KUKA KRL program: s1001_1.src

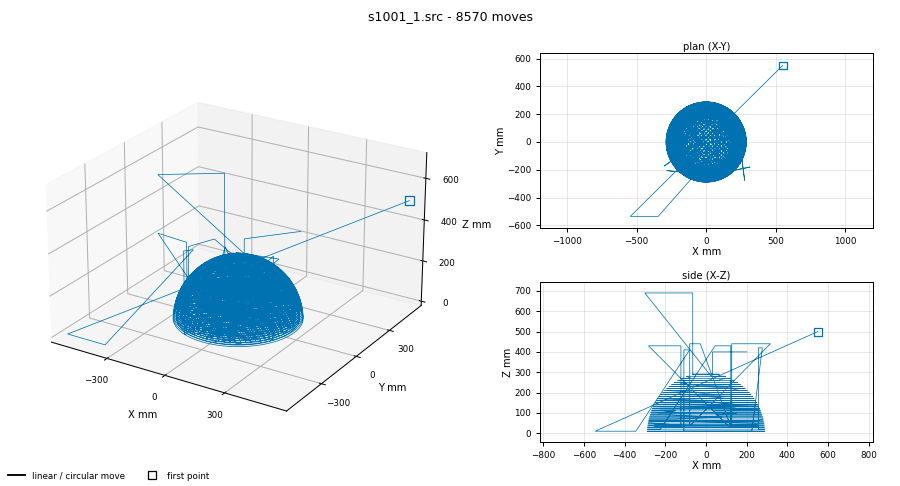
[picture p0: tool path of s1001_1.src, 8570 of 8571 moves have a stored position in this frame; points joined in program order, loops and branches not executed]
&ACCESS RVO
DEF s1001_1()
;TOOLPATH
PTP {A1 0,A2 -135,A3 135,A4 75,A5 30,A6 -65,E1 0,E2 0,E3 0,E4 0,E5 0,E6 0}
$VEL.CP=0.3
LIN {X 550.000,Y 550.000,Z 500.000,A 0.000,B 0.000,C 180.000,E1 0.000} C_DIS
;--------------------------------
;Part 1
;rapid-leaky
LIN {X -545.000,Y -535.000,Z 10.000,A 0.000,B 0.000,C 180.000,E1 0.000} C_DIS

EXTRUDER_STATE=TRUE
LIN {X -545.000,Y -535.000,Z 10.000,A 0.000,B 0.000,C 180.000,E1 0.000} C_DIS
;bead-prime
$VEL.CP=1
LIN {X -345.000,Y -535.000,Z 10.000,A 0.000,B 0.000,C 180.000,E1 0.000} C_DIS
$VEL.CP=0.3
LIN {X -345.000,Y -535.000,Z 10.000,A 0.000,B 0.000,C 180.000,E1 0.000} C_DIS

EXTRUDER_STATE=FALSE
LIN {X -80.274,Y -235.133,Z 410.000,A 0.000,B 0.000,C 180.000,E1 0.000} C_DIS
LIN {X -108.740,Y -267.377,Z 410.000,A 0.000,B 0.000,C 180.000,E1 0.000} C_DIS
LIN {X -108.740,Y -267.377,Z 10.000,A 0.000,B 0.000,C 180.000,E1 0.000} C_DIS
LIN {X -108.740,Y -267.377,Z 10.000,A 0.000,B 0.000,C 180.000,E1 0.000} C_DIS
EXTRUDER_STATE=TRUE

;bead-perimeter_outer
$VEL.CP=0.5
LIN {X -94.832,Y -272.621,Z 10.000,A 0.000,B 0.000,C 180.000,E1 0.000} C_DIS
LIN {X -80.672,Y -277.141,Z 10.000,A 0.000,B 0.000,C 180.000,E1 0.000} C_DIS
LIN {X -66.297,Y -280.927,Z 10.000,A 0.000,B 0.000,C 180.000,E1 0.000} C_DIS
LIN {X -51.748,Y -283.967,Z 10.000,A 0.000,B 0.000,C 180.000,E1 0.000} C_DIS
LIN {X -37.062,Y -286.255,Z 10.000,A 0.000,B 0.000,C 180.000,E1 0.000} C_DIS
LIN {X -22.276,Y -287.783,Z 10.000,A 0.000,B 0.000,C 180.000,E1 0.000} C_DIS
LIN {X -7.431,Y -288.549,Z 10.000,A 0.000,B 0.000,C 180.000,E1 0.000} C_DIS
LIN {X 7.431,Y -288.549,Z 10.000,A 0.000,B 0.000,C 180.000,E1 0.000} C_DIS
LIN {X 22.276,Y -287.783,Z 10.000,A 0.000,B 0.000,C 180.000,E1 0.000} C_DIS
LIN {X 37.062,Y -286.255,Z 10.000,A 0.000,B 0.000,C 180.000,E1 0.000} C_DIS
LIN {X 51.748,Y -283.967,Z 10.000,A 0.000,B 0.000,C 180.000,E1 0.000} C_DIS
LIN {X 66.297,Y -280.927,Z 10.000,A 0.000,B 0.000,C 180.000,E1 0.000} C_DIS
LIN {X 80.672,Y -277.141,Z 10.000,A 0.000,B 0.000,C 180.000,E1 0.000} C_DIS
LIN {X 94.832,Y -272.621,Z 10.000,A 0.000,B 0.000,C 180.000,E1 0.000} C_DIS
LIN {X 108.740,Y -267.377,Z 10.000,A 0.000,B 0.000,C 180.000,E1 0.000} C_DIS
LIN {X 122.360,Y -261.425,Z 10.000,A 0.000,B 0.000,C 180.000,E1 0.000} C_DIS
LIN {X 135.656,Y -254.780,Z 10.000,A 0.000,B 0.000,C 180.000,E1 0.000} C_DIS
LIN {X 148.592,Y -247.459,Z 10.000,A 0.000,B 0.000,C 180.000,E1 0.000} C_DIS
LIN {X 161.134,Y -239.481,Z 10.000,A 0.000,B 0.000,C 180.000,E1 0.000} C_DIS
LIN {X 173.248,Y -230.869,Z 10.000,A 0.000,B 0.000,C 180.000,E1 0.000} C_DIS
LIN {X 184.903,Y -221.644,Z 10.000,A 0.000,B 0.000,C 180.000,E1 0.000} C_DIS
LIN {X 196.068,Y -211.831,Z 10.000,A 0.000,B 0.000,C 180.000,E1 0.000} C_DIS
LIN {X 206.713,Y -201.457,Z 10.000,A 0.000,B 0.000,C 180.000,E1 0.000} C_DIS
LIN {X 216.810,Y -190.549,Z 10.000,A 0.000,B 0.000,C 180.000,E1 0.000} C_DIS
LIN {X 226.331,Y -179.135,Z 10.000,A 0.000,B 0.000,C 180.000,E1 0.000} C_DIS
LIN {X 235.253,Y -167.246,Z 10.000,A 0.000,B 0.000,C 180.000,E1 0.000} C_DIS
LIN {X 243.551,Y -154.914,Z 10.000,A 0.000,B 0.000,C 180.000,E1 0.000} C_DIS
LIN {X 251.203,Y -142.171,Z 10.000,A 0.000,B 0.000,C 180.000,E1 0.000} C_DIS
LIN {X 258.188,Y -129.051,Z 10.000,A 0.000,B 0.000,C 180.000,E1 0.000} C_DIS
LIN {X 264.490,Y -115.588,Z 10.000,A 0.000,B 0.000,C 180.000,E1 0.000} C_DIS
LIN {X 270.089,Y -101.820,Z 10.000,A 0.000,B 0.000,C 180.000,E1 0.000} C_DIS
LIN {X 274.972,Y -87.780,Z 10.000,A 0.000,B 0.000,C 180.000,E1 0.000} C_DIS
LIN {X 279.127,Y -73.509,Z 10.000,A 0.000,B 0.000,C 180.000,E1 0.000} C_DIS
LIN {X 282.541,Y -59.043,Z 10.000,A 0.000,B 0.000,C 180.000,E1 0.000} C_DIS
LIN {X 285.206,Y -44.419,Z 10.000,A 0.000,B 0.000,C 180.000,E1 0.000} C_DIS
LIN {X 287.114,Y -29.678,Z 10.000,A 0.000,B 0.000,C 180.000,E1 0.000} C_DIS
LIN {X 288.261,Y -14.860,Z 10.000,A 0.000,B 0.000,C 180.000,E1 0.000} C_DIS
LIN {X 288.644,Y 0.000,Z 10.000,A 0.000,B 0.000,C 180.000,E1 0.000} C_DIS
LIN {X 288.261,Y 14.859,Z 10.000,A 0.000,B 0.000,C 180.000,E1 0.000} C_DIS
LIN {X 287.114,Y 29.678,Z 10.000,A 0.000,B 0.000,C 180.000,E1 0.000} C_DIS
LIN {X 285.206,Y 44.419,Z 10.000,A 0.000,B 0.000,C 180.000,E1 0.000} C_DIS
LIN {X 282.541,Y 59.043,Z 10.000,A 0.000,B 0.000,C 180.000,E1 0.000} C_DIS
LIN {X 279.127,Y 73.509,Z 10.000,A 0.000,B 0.000,C 180.000,E1 0.000} C_DIS
LIN {X 274.972,Y 87.780,Z 10.000,A 0.000,B 0.000,C 180.000,E1 0.000} C_DIS
LIN {X 270.089,Y 101.820,Z 10.000,A 0.000,B 0.000,C 180.000,E1 0.000} C_DIS
LIN {X 264.490,Y 115.588,Z 10.000,A 0.000,B 0.000,C 180.000,E1 0.000} C_DIS
LIN {X 258.188,Y 129.051,Z 10.000,A 0.000,B 0.000,C 180.000,E1 0.000} C_DIS
LIN {X 251.203,Y 142.171,Z 10.000,A 0.000,B 0.000,C 180.000,E1 0.000} C_DIS
LIN {X 243.551,Y 154.914,Z 10.000,A 0.000,B 0.000,C 180.000,E1 0.000} C_DIS
LIN {X 235.253,Y 167.246,Z 10.000,A 0.000,B 0.000,C 180.000,E1 0.000} C_DIS
LIN {X 226.331,Y 179.135,Z 10.000,A 0.000,B 0.000,C 180.000,E1 0.000} C_DIS
LIN {X 216.810,Y 190.549,Z 10.000,A 0.000,B 0.000,C 180.000,E1 0.000} C_DIS
LIN {X 206.713,Y 201.457,Z 10.000,A 0.000,B 0.000,C 180.000,E1 0.000} C_DIS
LIN {X 196.068,Y 211.831,Z 10.000,A 0.000,B 0.000,C 180.000,E1 0.000} C_DIS
LIN {X 184.903,Y 221.644,Z 10.000,A 0.000,B 0.000,C 180.000,E1 0.000} C_DIS
LIN {X 173.248,Y 230.869,Z 10.000,A 0.000,B 0.000,C 180.000,E1 0.000} C_DIS
LIN {X 161.133,Y 239.482,Z 10.000,A 0.000,B 0.000,C 180.000,E1 0.000} C_DIS
LIN {X 148.592,Y 247.459,Z 10.000,A 0.000,B 0.000,C 180.000,E1 0.000} C_DIS
LIN {X 135.656,Y 254.780,Z 10.000,A 0.000,B 0.000,C 180.000,E1 0.000} C_DIS
LIN {X 122.360,Y 261.425,Z 10.000,A 0.000,B 0.000,C 180.000,E1 0.000} C_DIS
LIN {X 108.740,Y 267.377,Z 10.000,A 0.000,B 0.000,C 180.000,E1 0.000} C_DIS
LIN {X 94.832,Y 272.621,Z 10.000,A 0.000,B 0.000,C 180.000,E1 0.000} C_DIS
LIN {X 80.672,Y 277.141,Z 10.000,A 0.000,B 0.000,C 180.000,E1 0.000} C_DIS
LIN {X 66.297,Y 280.927,Z 10.000,A 0.000,B 0.000,C 180.000,E1 0.000} C_DIS
LIN {X 51.748,Y 283.967,Z 10.000,A 0.000,B 0.000,C 180.000,E1 0.000} C_DIS
LIN {X 37.062,Y 286.255,Z 10.000,A 0.000,B 0.000,C 180.000,E1 0.000} C_DIS
LIN {X 22.276,Y 287.783,Z 10.000,A 0.000,B 0.000,C 180.000,E1 0.000} C_DIS
LIN {X 7.431,Y 288.549,Z 10.000,A 0.000,B 0.000,C 180.000,E1 0.000} C_DIS
LIN {X -7.431,Y 288.549,Z 10.000,A 0.000,B 0.000,C 180.000,E1 0.000} C_DIS
LIN {X -22.276,Y 287.783,Z 10.000,A 0.000,B 0.000,C 180.000,E1 0.000} C_DIS
LIN {X -37.062,Y 286.255,Z 10.000,A 0.000,B 0.000,C 180.000,E1 0.000} C_DIS
LIN {X -51.748,Y 283.967,Z 10.000,A 0.000,B 0.000,C 180.000,E1 0.000} C_DIS
LIN {X -66.297,Y 280.927,Z 10.000,A 0.000,B 0.000,C 180.000,E1 0.000} C_DIS
LIN {X -80.672,Y 277.141,Z 10.000,A 0.000,B 0.000,C 180.000,E1 0.000} C_DIS
LIN {X -94.832,Y 272.621,Z 10.000,A 0.000,B 0.000,C 180.000,E1 0.000} C_DIS
LIN {X -108.740,Y 267.377,Z 10.000,A 0.000,B 0.000,C 180.000,E1 0.000} C_DIS
LIN {X -122.360,Y 261.425,Z 10.000,A 0.000,B 0.000,C 180.000,E1 0.000} C_DIS
LIN {X -135.656,Y 254.780,Z 10.000,A 0.000,B 0.000,C 180.000,E1 0.000} C_DIS
LIN {X -148.592,Y 247.459,Z 10.000,A 0.000,B 0.000,C 180.000,E1 0.000} C_DIS
LIN {X -161.134,Y 239.481,Z 10.000,A 0.000,B 0.000,C 180.000,E1 0.000} C_DIS
LIN {X -173.248,Y 230.869,Z 10.000,A 0.000,B 0.000,C 180.000,E1 0.000} C_DIS
LIN {X -184.903,Y 221.644,Z 10.000,A 0.000,B 0.000,C 180.000,E1 0.000} C_DIS
LIN {X -196.068,Y 211.831,Z 10.000,A 0.000,B 0.000,C 180.000,E1 0.000} C_DIS
LIN {X -206.713,Y 201.457,Z 10.000,A 0.000,B 0.000,C 180.000,E1 0.000} C_DIS
LIN {X -216.810,Y 190.549,Z 10.000,A 0.000,B 0.000,C 180.000,E1 0.000} C_DIS
LIN {X -226.331,Y 179.135,Z 10.000,A 0.000,B 0.000,C 180.000,E1 0.000} C_DIS
LIN {X -235.253,Y 167.246,Z 10.000,A 0.000,B 0.000,C 180.000,E1 0.000} C_DIS
LIN {X -243.551,Y 154.914,Z 10.000,A 0.000,B 0.000,C 180.000,E1 0.000} C_DIS
LIN {X -251.203,Y 142.171,Z 10.000,A 0.000,B 0.000,C 180.000,E1 0.000} C_DIS
LIN {X -258.188,Y 129.051,Z 10.000,A 0.000,B 0.000,C 180.000,E1 0.000} C_DIS
LIN {X -264.490,Y 115.588,Z 10.000,A 0.000,B 0.000,C 180.000,E1 0.000} C_DIS
LIN {X -270.089,Y 101.820,Z 10.000,A 0.000,B 0.000,C 180.000,E1 0.000} C_DIS
LIN {X -274.972,Y 87.780,Z 10.000,A 0.000,B 0.000,C 180.000,E1 0.000} C_DIS
LIN {X -279.127,Y 73.509,Z 10.000,A 0.000,B 0.000,C 180.000,E1 0.000} C_DIS
LIN {X -282.541,Y 59.043,Z 10.000,A 0.000,B 0.000,C 180.000,E1 0.000} C_DIS
LIN {X -285.206,Y 44.419,Z 10.000,A 0.000,B 0.000,C 180.000,E1 0.000} C_DIS
LIN {X -287.114,Y 29.678,Z 10.000,A 0.000,B 0.000,C 180.000,E1 0.000} C_DIS
LIN {X -287.873,Y 19.878,Z 10.000,A 0.000,B 0.000,C 180.000,E1 0.000} C_DIS
LIN {X -288.261,Y 14.860,Z 10.000,A 0.000,B 0.000,C 180.000,E1 0.000} C_DIS
LIN {X -288.644,Y 0.000,Z 10.000,A 0.000,B 0.000,C 180.000,E1 0.000} C_DIS
LIN {X -288.261,Y -14.859,Z 10.000,A 0.000,B 0.000,C 180.000,E1 0.000} C_DIS
LIN {X -287.114,Y -29.678,Z 10.000,A 0.000,B 0.000,C 180.000,E1 0.000} C_DIS
LIN {X -285.206,Y -44.419,Z 10.000,A 0.000,B 0.000,C 180.000,E1 0.000} C_DIS
LIN {X -282.541,Y -59.043,Z 10.000,A 0.000,B 0.000,C 180.000,E1 0.000} C_DIS
LIN {X -279.127,Y -73.509,Z 10.000,A 0.000,B 0.000,C 180.000,E1 0.000} C_DIS
LIN {X -274.972,Y -87.780,Z 10.000,A 0.000,B 0.000,C 180.000,E1 0.000} C_DIS
LIN {X -270.089,Y -101.820,Z 10.000,A 0.000,B 0.000,C 180.000,E1 0.000} C_DIS
LIN {X -264.490,Y -115.588,Z 10.000,A 0.000,B 0.000,C 180.000,E1 0.000} C_DIS
LIN {X -258.188,Y -129.051,Z 10.000,A 0.000,B 0.000,C 180.000,E1 0.000} C_DIS
LIN {X -251.203,Y -142.171,Z 10.000,A 0.000,B 0.000,C 180.000,E1 0.000} C_DIS
LIN {X -243.551,Y -154.914,Z 10.000,A 0.000,B 0.000,C 180.000,E1 0.000} C_DIS
LIN {X -235.253,Y -167.246,Z 10.000,A 0.000,B 0.000,C 180.000,E1 0.000} C_DIS
LIN {X -226.331,Y -179.135,Z 10.000,A 0.000,B 0.000,C 180.000,E1 0.000} C_DIS
LIN {X -216.810,Y -190.549,Z 10.000,A 0.000,B 0.000,C 180.000,E1 0.000} C_DIS
LIN {X -206.713,Y -201.457,Z 10.000,A 0.000,B 0.000,C 180.000,E1 0.000} C_DIS
LIN {X -196.068,Y -211.831,Z 10.000,A 0.000,B 0.000,C 180.000,E1 0.000} C_DIS
LIN {X -184.903,Y -221.644,Z 10.000,A 0.000,B 0.000,C 180.000,E1 0.000} C_DIS
LIN {X -173.248,Y -230.869,Z 10.000,A 0.000,B 0.000,C 180.000,E1 0.000} C_DIS
LIN {X -161.133,Y -239.482,Z 10.000,A 0.000,B 0.000,C 180.000,E1 0.000} C_DIS
LIN {X -148.592,Y -247.459,Z 10.000,A 0.000,B 0.000,C 180.000,E1 0.000} C_DIS
LIN {X -135.656,Y -254.780,Z 10.000,A 0.000,B 0.000,C 180.000,E1 0.000} C_DIS
LIN {X -122.360,Y -261.425,Z 10.000,A 0.000,B 0.000,C 180.000,E1 0.000} C_DIS
LIN {X -108.740,Y -267.377,Z 10.000,A 0.000,B 0.000,C 180.000,E1 0.000} C_DIS
;rapid-leaky
$VEL.CP=0.3
LIN {X -102.884,Y -252.978,Z 10.000,A 0.000,B 0.000,C 180.000,E1 0.000} C_DIS
;bead-perimeter_inner
$VEL.CP=0.5
LIN {X -89.725,Y -257.938,Z 10.000,A 0.000,B 0.000,C 180.000,E1 0.000} C_DIS
LIN {X -76.327,Y -262.215,Z 10.000,A 0.000,B 0.000,C 180.000,E1 0.000} C_DIS
LIN {X -62.727,Y -265.798,Z 10.000,A 0.000,B 0.000,C 180.000,E1 0.000} C_DIS
LIN {X -48.961,Y -268.674,Z 10.000,A 0.000,B 0.000,C 180.000,E1 0.000} C_DIS
LIN {X -35.066,Y -270.839,Z 10.000,A 0.000,B 0.000,C 180.000,E1 0.000} C_DIS
LIN {X -21.076,Y -272.284,Z 10.000,A 0.000,B 0.000,C 180.000,E1 0.000} C_DIS
LIN {X -7.030,Y -273.009,Z 10.000,A 0.000,B 0.000,C 180.000,E1 0.000} C_DIS
LIN {X 7.030,Y -273.009,Z 10.000,A 0.000,B 0.000,C 180.000,E1 0.000} C_DIS
LIN {X 21.076,Y -272.284,Z 10.000,A 0.000,B 0.000,C 180.000,E1 0.000} C_DIS
LIN {X 35.066,Y -270.839,Z 10.000,A 0.000,B 0.000,C 180.000,E1 0.000} C_DIS
LIN {X 48.961,Y -268.674,Z 10.000,A 0.000,B 0.000,C 180.000,E1 0.000} C_DIS
LIN {X 62.727,Y -265.798,Z 10.000,A 0.000,B 0.000,C 180.000,E1 0.000} C_DIS
LIN {X 76.327,Y -262.215,Z 10.000,A 0.000,B 0.000,C 180.000,E1 0.000} C_DIS
LIN {X 89.725,Y -257.938,Z 10.000,A 0.000,B 0.000,C 180.000,E1 0.000} C_DIS
LIN {X 102.884,Y -252.978,Z 10.000,A 0.000,B 0.000,C 180.000,E1 0.000} C_DIS
LIN {X 115.771,Y -247.346,Z 10.000,A 0.000,B 0.000,C 180.000,E1 0.000} C_DIS
LIN {X 128.350,Y -241.059,Z 10.000,A 0.000,B 0.000,C 180.000,E1 0.000} C_DIS
LIN {X 140.590,Y -234.132,Z 10.000,A 0.000,B 0.000,C 180.000,E1 0.000} C_DIS
LIN {X 152.456,Y -226.584,Z 10.000,A 0.000,B 0.000,C 180.000,E1 0.000} C_DIS
LIN {X 163.917,Y -218.436,Z 10.000,A 0.000,B 0.000,C 180.000,E1 0.000} C_DIS
LIN {X 174.944,Y -209.707,Z 10.000,A 0.000,B 0.000,C 180.000,E1 0.000} C_DIS
LIN {X 185.508,Y -200.423,Z 10.000,A 0.000,B 0.000,C 180.000,E1 0.000} C_DIS
LIN {X 195.581,Y -190.607,Z 10.000,A 0.000,B 0.000,C 180.000,E1 0.000} C_DIS
LIN {X 205.133,Y -180.287,Z 10.000,A 0.000,B 0.000,C 180.000,E1 0.000} C_DIS
LIN {X 214.142,Y -169.487,Z 10.000,A 0.000,B 0.000,C 180.000,E1 0.000} C_DIS
LIN {X 222.584,Y -158.239,Z 10.000,A 0.000,B 0.000,C 180.000,E1 0.000} C_DIS
LIN {X 230.434,Y -146.571,Z 10.000,A 0.000,B 0.000,C 180.000,E1 0.000} C_DIS
LIN {X 237.674,Y -134.515,Z 10.000,A 0.000,B 0.000,C 180.000,E1 0.000} C_DIS
LIN {X 244.283,Y -122.100,Z 10.000,A 0.000,B 0.000,C 180.000,E1 0.000} C_DIS
LIN {X 250.245,Y -109.363,Z 10.000,A 0.000,B 0.000,C 180.000,E1 0.000} C_DIS
LIN {X 255.543,Y -96.337,Z 10.000,A 0.000,B 0.000,C 180.000,E1 0.000} C_DIS
LIN {X 260.163,Y -83.053,Z 10.000,A 0.000,B 0.000,C 180.000,E1 0.000} C_DIS
LIN {X 264.094,Y -69.550,Z 10.000,A 0.000,B 0.000,C 180.000,E1 0.000} C_DIS
LIN {X 267.325,Y -55.863,Z 10.000,A 0.000,B 0.000,C 180.000,E1 0.000} C_DIS
LIN {X 269.846,Y -42.027,Z 10.000,A 0.000,B 0.000,C 180.000,E1 0.000} C_DIS
LIN {X 271.651,Y -28.079,Z 10.000,A 0.000,B 0.000,C 180.000,E1 0.000} C_DIS
LIN {X 272.737,Y -14.060,Z 10.000,A 0.000,B 0.000,C 180.000,E1 0.000} C_DIS
LIN {X 273.099,Y 0.000,Z 10.000,A 0.000,B 0.000,C 180.000,E1 0.000} C_DIS
LIN {X 272.737,Y 14.059,Z 10.000,A 0.000,B 0.000,C 180.000,E1 0.000} C_DIS
LIN {X 271.651,Y 28.080,Z 10.000,A 0.000,B 0.000,C 180.000,E1 0.000} C_DIS
LIN {X 269.846,Y 42.027,Z 10.000,A 0.000,B 0.000,C 180.000,E1 0.000} C_DIS
LIN {X 267.325,Y 55.863,Z 10.000,A 0.000,B 0.000,C 180.000,E1 0.000} C_DIS
LIN {X 264.094,Y 69.550,Z 10.000,A 0.000,B 0.000,C 180.000,E1 0.000} C_DIS
LIN {X 260.163,Y 83.053,Z 10.000,A 0.000,B 0.000,C 180.000,E1 0.000} C_DIS
LIN {X 255.543,Y 96.337,Z 10.000,A 0.000,B 0.000,C 180.000,E1 0.000} C_DIS
LIN {X 250.245,Y 109.363,Z 10.000,A 0.000,B 0.000,C 180.000,E1 0.000} C_DIS
LIN {X 244.283,Y 122.100,Z 10.000,A 0.000,B 0.000,C 180.000,E1 0.000} C_DIS
LIN {X 237.674,Y 134.515,Z 10.000,A 0.000,B 0.000,C 180.000,E1 0.000} C_DIS
LIN {X 230.434,Y 146.571,Z 10.000,A 0.000,B 0.000,C 180.000,E1 0.000} C_DIS
LIN {X 222.584,Y 158.239,Z 10.000,A 0.000,B 0.000,C 180.000,E1 0.000} C_DIS
LIN {X 214.142,Y 169.487,Z 10.000,A 0.000,B 0.000,C 180.000,E1 0.000} C_DIS
LIN {X 205.133,Y 180.287,Z 10.000,A 0.000,B 0.000,C 180.000,E1 0.000} C_DIS
LIN {X 195.581,Y 190.607,Z 10.000,A 0.000,B 0.000,C 180.000,E1 0.000} C_DIS
LIN {X 185.508,Y 200.423,Z 10.000,A 0.000,B 0.000,C 180.000,E1 0.000} C_DIS
LIN {X 174.944,Y 209.707,Z 10.000,A 0.000,B 0.000,C 180.000,E1 0.000} C_DIS
LIN {X 163.918,Y 218.436,Z 10.000,A 0.000,B 0.000,C 180.000,E1 0.000} C_DIS
LIN {X 152.456,Y 226.584,Z 10.000,A 0.000,B 0.000,C 180.000,E1 0.000} C_DIS
LIN {X 140.590,Y 234.132,Z 10.000,A 0.000,B 0.000,C 180.000,E1 0.000} C_DIS
LIN {X 128.350,Y 241.059,Z 10.000,A 0.000,B 0.000,C 180.000,E1 0.000} C_DIS
LIN {X 115.771,Y 247.346,Z 10.000,A 0.000,B 0.000,C 180.000,E1 0.000} C_DIS
LIN {X 102.884,Y 252.978,Z 10.000,A 0.000,B 0.000,C 180.000,E1 0.000} C_DIS
LIN {X 89.725,Y 257.938,Z 10.000,A 0.000,B 0.000,C 180.000,E1 0.000} C_DIS
LIN {X 76.327,Y 262.215,Z 10.000,A 0.000,B 0.000,C 180.000,E1 0.000} C_DIS
LIN {X 62.727,Y 265.798,Z 10.000,A 0.000,B 0.000,C 180.000,E1 0.000} C_DIS
LIN {X 48.961,Y 268.674,Z 10.000,A 0.000,B 0.000,C 180.000,E1 0.000} C_DIS
LIN {X 35.066,Y 270.839,Z 10.000,A 0.000,B 0.000,C 180.000,E1 0.000} C_DIS
LIN {X 21.076,Y 272.284,Z 10.000,A 0.000,B 0.000,C 180.000,E1 0.000} C_DIS
LIN {X 7.030,Y 273.009,Z 10.000,A 0.000,B 0.000,C 180.000,E1 0.000} C_DIS
LIN {X -7.030,Y 273.009,Z 10.000,A 0.000,B 0.000,C 180.000,E1 0.000} C_DIS
LIN {X -21.076,Y 272.284,Z 10.000,A 0.000,B 0.000,C 180.000,E1 0.000} C_DIS
LIN {X -35.066,Y 270.839,Z 10.000,A 0.000,B 0.000,C 180.000,E1 0.000} C_DIS
LIN {X -48.961,Y 268.674,Z 10.000,A 0.000,B 0.000,C 180.000,E1 0.000} C_DIS
LIN {X -62.727,Y 265.798,Z 10.000,A 0.000,B 0.000,C 180.000,E1 0.000} C_DIS
LIN {X -76.327,Y 262.215,Z 10.000,A 0.000,B 0.000,C 180.000,E1 0.000} C_DIS
LIN {X -89.725,Y 257.938,Z 10.000,A 0.000,B 0.000,C 180.000,E1 0.000} C_DIS
LIN {X -102.884,Y 252.978,Z 10.000,A 0.000,B 0.000,C 180.000,E1 0.000} C_DIS
LIN {X -115.771,Y 247.346,Z 10.000,A 0.000,B 0.000,C 180.000,E1 0.000} C_DIS
LIN {X -128.350,Y 241.059,Z 10.000,A 0.000,B 0.000,C 180.000,E1 0.000} C_DIS
LIN {X -140.590,Y 234.132,Z 10.000,A 0.000,B 0.000,C 180.000,E1 0.000} C_DIS
LIN {X -152.456,Y 226.584,Z 10.000,A 0.000,B 0.000,C 180.000,E1 0.000} C_DIS
LIN {X -163.917,Y 218.436,Z 10.000,A 0.000,B 0.000,C 180.000,E1 0.000} C_DIS
LIN {X -174.944,Y 209.707,Z 10.000,A 0.000,B 0.000,C 180.000,E1 0.000} C_DIS
LIN {X -185.508,Y 200.423,Z 10.000,A 0.000,B 0.000,C 180.000,E1 0.000} C_DIS
LIN {X -195.581,Y 190.607,Z 10.000,A 0.000,B 0.000,C 180.000,E1 0.000} C_DIS
LIN {X -205.133,Y 180.287,Z 10.000,A 0.000,B 0.000,C 180.000,E1 0.000} C_DIS
LIN {X -214.142,Y 169.487,Z 10.000,A 0.000,B 0.000,C 180.000,E1 0.000} C_DIS
LIN {X -222.584,Y 158.239,Z 10.000,A 0.000,B 0.000,C 180.000,E1 0.000} C_DIS
LIN {X -230.434,Y 146.571,Z 10.000,A 0.000,B 0.000,C 180.000,E1 0.000} C_DIS
LIN {X -237.674,Y 134.515,Z 10.000,A 0.000,B 0.000,C 180.000,E1 0.000} C_DIS
LIN {X -244.283,Y 122.100,Z 10.000,A 0.000,B 0.000,C 180.000,E1 0.000} C_DIS
LIN {X -250.245,Y 109.363,Z 10.000,A 0.000,B 0.000,C 180.000,E1 0.000} C_DIS
LIN {X -255.543,Y 96.337,Z 10.000,A 0.000,B 0.000,C 180.000,E1 0.000} C_DIS
LIN {X -260.163,Y 83.053,Z 10.000,A 0.000,B 0.000,C 180.000,E1 0.000} C_DIS
LIN {X -264.094,Y 69.550,Z 10.000,A 0.000,B 0.000,C 180.000,E1 0.000} C_DIS
LIN {X -267.325,Y 55.863,Z 10.000,A 0.000,B 0.000,C 180.000,E1 0.000} C_DIS
LIN {X -269.846,Y 42.027,Z 10.000,A 0.000,B 0.000,C 180.000,E1 0.000} C_DIS
LIN {X -271.651,Y 28.079,Z 10.000,A 0.000,B 0.000,C 180.000,E1 0.000} C_DIS
LIN {X -272.380,Y 18.678,Z 10.000,A 0.000,B 0.000,C 180.000,E1 0.000} C_DIS
LIN {X -272.737,Y 14.060,Z 10.000,A 0.000,B 0.000,C 180.000,E1 0.000} C_DIS
LIN {X -273.099,Y 0.000,Z 10.000,A 0.000,B 0.000,C 180.000,E1 0.000} C_DIS
LIN {X -272.737,Y -14.059,Z 10.000,A 0.000,B 0.000,C 180.000,E1 0.000} C_DIS
LIN {X -271.651,Y -28.080,Z 10.000,A 0.000,B 0.000,C 180.000,E1 0.000} C_DIS
LIN {X -269.846,Y -42.027,Z 10.000,A 0.000,B 0.000,C 180.000,E1 0.000} C_DIS
LIN {X -267.325,Y -55.863,Z 10.000,A 0.000,B 0.000,C 180.000,E1 0.000} C_DIS
LIN {X -264.094,Y -69.550,Z 10.000,A 0.000,B 0.000,C 180.000,E1 0.000} C_DIS
LIN {X -260.163,Y -83.053,Z 10.000,A 0.000,B 0.000,C 180.000,E1 0.000} C_DIS
LIN {X -255.543,Y -96.337,Z 10.000,A 0.000,B 0.000,C 180.000,E1 0.000} C_DIS
LIN {X -250.245,Y -109.363,Z 10.000,A 0.000,B 0.000,C 180.000,E1 0.000} C_DIS
LIN {X -244.283,Y -122.100,Z 10.000,A 0.000,B 0.000,C 180.000,E1 0.000} C_DIS
LIN {X -237.674,Y -134.515,Z 10.000,A 0.000,B 0.000,C 180.000,E1 0.000} C_DIS
LIN {X -230.434,Y -146.571,Z 10.000,A 0.000,B 0.000,C 180.000,E1 0.000} C_DIS
LIN {X -222.584,Y -158.239,Z 10.000,A 0.000,B 0.000,C 180.000,E1 0.000} C_DIS
LIN {X -214.142,Y -169.487,Z 10.000,A 0.000,B 0.000,C 180.000,E1 0.000} C_DIS
LIN {X -205.133,Y -180.287,Z 10.000,A 0.000,B 0.000,C 180.000,E1 0.000} C_DIS
LIN {X -195.581,Y -190.607,Z 10.000,A 0.000,B 0.000,C 180.000,E1 0.000} C_DIS
LIN {X -185.508,Y -200.423,Z 10.000,A 0.000,B 0.000,C 180.000,E1 0.000} C_DIS
LIN {X -174.944,Y -209.707,Z 10.000,A 0.000,B 0.000,C 180.000,E1 0.000} C_DIS
LIN {X -163.918,Y -218.436,Z 10.000,A 0.000,B 0.000,C 180.000,E1 0.000} C_DIS
LIN {X -152.456,Y -226.584,Z 10.000,A 0.000,B 0.000,C 180.000,E1 0.000} C_DIS
LIN {X -140.590,Y -234.132,Z 10.000,A 0.000,B 0.000,C 180.000,E1 0.000} C_DIS
LIN {X -128.350,Y -241.059,Z 10.000,A 0.000,B 0.000,C 180.000,E1 0.000} C_DIS
LIN {X -115.771,Y -247.346,Z 10.000,A 0.000,B 0.000,C 180.000,E1 0.000} C_DIS
LIN {X -102.884,Y -252.978,Z 10.000,A 0.000,B 0.000,C 180.000,E1 0.000} C_DIS
;rapid-leaky
$VEL.CP=0.3
LIN {X -225.167,Y -120.215,Z 10.000,A 0.000,B 0.000,C 180.000,E1 0.000} C_DIS
;bead-solid_infill
$VEL.CP=0.5
LIN {X -120.009,Y -225.372,Z 10.000,A 0.000,B 0.000,C 180.000,E1 0.000} C_DIS
LIN {X -120.000,Y -225.377,Z 10.000,A 0.000,B 0.000,C 180.000,E1 0.000} C_DIS
LIN {X -108.240,Y -231.255,Z 10.000,A 0.000,B 0.000,C 180.000,E1 0.000} C_DIS
LIN {X -96.191,Y -236.521,Z 10.000,A 0.000,B 0.000,C 180.000,E1 0.000} C_DIS
LIN {X -83.888,Y -241.159,Z 10.000,A 0.000,B 0.000,C 180.000,E1 0.000} C_DIS
LIN {X -71.361,Y -245.157,Z 10.000,A 0.000,B 0.000,C 180.000,E1 0.000} C_DIS
LIN {X -67.922,Y -246.063,Z 10.000,A 0.000,B 0.000,C 180.000,E1 0.000} C_DIS
LIN {X -246.073,Y -67.912,Z 10.000,A 0.000,B 0.000,C 180.000,E1 0.000} C_DIS
LIN {X -246.914,Y -65.025,Z 10.000,A 0.000,B 0.000,C 180.000,E1 0.000} C_DIS
LIN {X -249.934,Y -52.229,Z 10.000,A 0.000,B 0.000,C 180.000,E1 0.000} C_DIS
LIN {X -252.291,Y -39.293,Z 10.000,A 0.000,B 0.000,C 180.000,E1 0.000} C_DIS
LIN {X -253.629,Y -28.961,Z 10.000,A 0.000,B 0.000,C 180.000,E1 0.000} C_DIS
LIN {X -28.977,Y -253.613,Z 10.000,A 0.000,B 0.000,C 180.000,E1 0.000} C_DIS
LIN {X -19.705,Y -254.571,Z 10.000,A 0.000,B 0.000,C 180.000,E1 0.000} C_DIS
LIN {X -6.571,Y -255.249,Z 10.000,A 0.000,B 0.000,C 180.000,E1 0.000} C_DIS
LIN {X 4.054,Y -255.249,Z 10.000,A 0.000,B 0.000,C 180.000,E1 0.000} C_DIS
LIN {X -255.229,Y 4.034,Z 10.000,A 0.000,B 0.000,C 180.000,E1 0.000} C_DIS
LIN {X -254.994,Y 13.146,Z 10.000,A 0.000,B 0.000,C 180.000,E1 0.000} C_DIS
LIN {X -254.673,Y 17.303,Z 10.000,A 0.000,B 0.000,C 180.000,E1 0.000} C_DIS
LIN {X -253.980,Y 26.252,Z 10.000,A 0.000,B 0.000,C 180.000,E1 0.000} C_DIS
LIN {X -253.071,Y 33.272,Z 10.000,A 0.000,B 0.000,C 180.000,E1 0.000} C_DIS
LIN {X 33.335,Y -253.134,Z 10.000,A 0.000,B 0.000,C 180.000,E1 0.000} C_DIS
LIN {X 45.776,Y -251.196,Z 10.000,A 0.000,B 0.000,C 180.000,E1 0.000} C_DIS
LIN {X 58.646,Y -248.507,Z 10.000,A 0.000,B 0.000,C 180.000,E1 0.000} C_DIS
LIN {X 59.800,Y -248.203,Z 10.000,A 0.000,B 0.000,C 180.000,E1 0.000} C_DIS
LIN {X -248.158,Y 59.754,Z 10.000,A 0.000,B 0.000,C 180.000,E1 0.000} C_DIS
LIN {X -246.914,Y 65.025,Z 10.000,A 0.000,B 0.000,C 180.000,E1 0.000} C_DIS
LIN {X -243.239,Y 77.651,Z 10.000,A 0.000,B 0.000,C 180.000,E1 0.000} C_DIS
LIN {X -241.025,Y 84.016,Z 10.000,A 0.000,B 0.000,C 180.000,E1 0.000} C_DIS
LIN {X 84.079,Y -241.087,Z 10.000,A 0.000,B 0.000,C 180.000,E1 0.000} C_DIS
LIN {X 96.191,Y -236.521,Z 10.000,A 0.000,B 0.000,C 180.000,E1 0.000} C_DIS
LIN {X 106.433,Y -232.045,Z 10.000,A 0.000,B 0.000,C 180.000,E1 0.000} C_DIS
LIN {X -232.020,Y 106.407,Z 10.000,A 0.000,B 0.000,C 180.000,E1 0.000} C_DIS
LIN {X -228.392,Y 114.157,Z 10.000,A 0.000,B 0.000,C 180.000,E1 0.000} C_DIS
LIN {X -222.212,Y 125.764,Z 10.000,A 0.000,B 0.000,C 180.000,E1 0.000} C_DIS
LIN {X -221.375,Y 127.158,Z 10.000,A 0.000,B 0.000,C 180.000,E1 0.000} C_DIS
LIN {X 127.127,Y -221.344,Z 10.000,A 0.000,B 0.000,C 180.000,E1 0.000} C_DIS
LIN {X 131.444,Y -218.900,Z 10.000,A 0.000,B 0.000,C 180.000,E1 0.000} C_DIS
LIN {X 142.538,Y -211.844,Z 10.000,A 0.000,B 0.000,C 180.000,E1 0.000} C_DIS
LIN {X 146.328,Y -209.149,Z 10.000,A 0.000,B 0.000,C 180.000,E1 0.000} C_DIS
LIN {X -209.175,Y 146.353,Z 10.000,A 0.000,B 0.000,C 180.000,E1 0.000} C_DIS
LIN {X -208.104,Y 147.945,Z 10.000,A 0.000,B 0.000,C 180.000,E1 0.000} C_DIS
LIN {X -200.212,Y 158.462,Z 10.000,A 0.000,B 0.000,C 180.000,E1 0.000} C_DIS
LIN {X -195.516,Y 164.090,Z 10.000,A 0.000,B 0.000,C 180.000,E1 0.000} C_DIS
LIN {X 164.136,Y -195.562,Z 10.000,A 0.000,B 0.000,C 180.000,E1 0.000} C_DIS
LIN {X 173.441,Y -187.384,Z 10.000,A 0.000,B 0.000,C 180.000,E1 0.000} C_DIS
LIN {X 180.487,Y -180.517,Z 10.000,A 0.000,B 0.000,C 180.000,E1 0.000} C_DIS
LIN {X -180.518,Y 180.487,Z 10.000,A 0.000,B 0.000,C 180.000,E1 0.000} C_DIS
LIN {X -173.441,Y 187.384,Z 10.000,A 0.000,B 0.000,C 180.000,E1 0.000} C_DIS
LIN {X -164.169,Y 195.534,Z 10.000,A 0.000,B 0.000,C 180.000,E1 0.000} C_DIS
LIN {X 195.489,Y -164.123,Z 10.000,A 0.000,B 0.000,C 180.000,E1 0.000} C_DIS
LIN {X 200.212,Y -158.462,Z 10.000,A 0.000,B 0.000,C 180.000,E1 0.000} C_DIS
LIN {X 208.104,Y -147.945,Z 10.000,A 0.000,B 0.000,C 180.000,E1 0.000} C_DIS
LIN {X 209.150,Y -146.390,Z 10.000,A 0.000,B 0.000,C 180.000,E1 0.000} C_DIS
LIN {X -146.364,Y 209.124,Z 10.000,A 0.000,B 0.000,C 180.000,E1 0.000} C_DIS
LIN {X -142.538,Y 211.844,Z 10.000,A 0.000,B 0.000,C 180.000,E1 0.000} C_DIS
LIN {X -131.444,Y 218.900,Z 10.000,A 0.000,B 0.000,C 180.000,E1 0.000} C_DIS
LIN {X -127.166,Y 221.322,Z 10.000,A 0.000,B 0.000,C 180.000,E1 0.000} C_DIS
LIN {X 221.352,Y -127.196,Z 10.000,A 0.000,B 0.000,C 180.000,E1 0.000} C_DIS
LIN {X 222.212,Y -125.764,Z 10.000,A 0.000,B 0.000,C 180.000,E1 0.000} C_DIS
LIN {X 228.392,Y -114.157,Z 10.000,A 0.000,B 0.000,C 180.000,E1 0.000} C_DIS
LIN {X 232.000,Y -106.448,Z 10.000,A 0.000,B 0.000,C 180.000,E1 0.000} C_DIS
LIN {X -106.475,Y 232.026,Z 10.000,A 0.000,B 0.000,C 180.000,E1 0.000} C_DIS
LIN {X -96.191,Y 236.521,Z 10.000,A 0.000,B 0.000,C 180.000,E1 0.000} C_DIS
LIN {X -84.123,Y 241.070,Z 10.000,A 0.000,B 0.000,C 180.000,E1 0.000} C_DIS
LIN {X 241.009,Y -84.061,Z 10.000,A 0.000,B 0.000,C 180.000,E1 0.000} C_DIS
LIN {X 243.239,Y -77.651,Z 10.000,A 0.000,B 0.000,C 180.000,E1 0.000} C_DIS
LIN {X 244.964,Y -71.725,Z 10.000,A 0.000,B 0.000,C 180.000,E1 0.000} C_DIS
LIN {X 246.914,Y -65.025,Z 10.000,A 0.000,B 0.000,C 180.000,E1 0.000} C_DIS
LIN {X 248.146,Y -59.803,Z 10.000,A 0.000,B 0.000,C 180.000,E1 0.000} C_DIS
LIN {X -59.848,Y 248.190,Z 10.000,A 0.000,B 0.000,C 180.000,E1 0.000} C_DIS
LIN {X -58.646,Y 248.507,Z 10.000,A 0.000,B 0.000,C 180.000,E1 0.000} C_DIS
LIN {X -45.776,Y 251.196,Z 10.000,A 0.000,B 0.000,C 180.000,E1 0.000} C_DIS
LIN {X -33.388,Y 253.126,Z 10.000,A 0.000,B 0.000,C 180.000,E1 0.000} C_DIS
LIN {X 253.064,Y -33.325,Z 10.000,A 0.000,B 0.000,C 180.000,E1 0.000} C_DIS
LIN {X 253.980,Y -26.253,Z 10.000,A 0.000,B 0.000,C 180.000,E1 0.000} C_DIS
LIN {X 255.503,Y -6.574,Z 10.000,A 0.000,B 0.000,C 180.000,E1 0.000} C_DIS
LIN {X 255.444,Y -4.310,Z 10.000,A 0.000,B 0.000,C 180.000,E1 0.000} C_DIS
LIN {X -4.115,Y 255.249,Z 10.000,A 0.000,B 0.000,C 180.000,E1 0.000} C_DIS
LIN {X 6.571,Y 255.249,Z 10.000,A 0.000,B 0.000,C 180.000,E1 0.000} C_DIS
LIN {X 19.705,Y 254.571,Z 10.000,A 0.000,B 0.000,C 180.000,E1 0.000} C_DIS
LIN {X 28.909,Y 253.620,Z 10.000,A 0.000,B 0.000,C 180.000,E1 0.000} C_DIS
LIN {X 253.638,Y 28.892,Z 10.000,A 0.000,B 0.000,C 180.000,E1 0.000} C_DIS
LIN {X 252.291,Y 39.293,Z 10.000,A 0.000,B 0.000,C 180.000,E1 0.000} C_DIS
LIN {X 249.934,Y 52.229,Z 10.000,A 0.000,B 0.000,C 180.000,E1 0.000} C_DIS
LIN {X 246.914,Y 65.025,Z 10.000,A 0.000,B 0.000,C 180.000,E1 0.000} C_DIS
LIN {X 246.098,Y 67.827,Z 10.000,A 0.000,B 0.000,C 180.000,E1 0.000} C_DIS
LIN {X 67.840,Y 246.085,Z 10.000,A 0.000,B 0.000,C 180.000,E1 0.000} C_DIS
LIN {X 71.361,Y 245.157,Z 10.000,A 0.000,B 0.000,C 180.000,E1 0.000} C_DIS
LIN {X 83.888,Y 241.159,Z 10.000,A 0.000,B 0.000,C 180.000,E1 0.000} C_DIS
LIN {X 96.191,Y 236.521,Z 10.000,A 0.000,B 0.000,C 180.000,E1 0.000} C_DIS
LIN {X 108.240,Y 231.255,Z 10.000,A 0.000,B 0.000,C 180.000,E1 0.000} C_DIS
LIN {X 119.887,Y 225.434,Z 10.000,A 0.000,B 0.000,C 180.000,E1 0.000} C_DIS
LIN {X 225.236,Y 120.085,Z 10.000,A 0.000,B 0.000,C 180.000,E1 0.000} C_DIS
$VEL.CP=0.3
LIN {X 225.236,Y 120.085,Z 10.000,A 0.000,B 0.000,C 180.000,E1 0.000} C_DIS
EXTRUDER_STATE=FALSE

LIN {X 277.036,Y -276.547,Z 420.000,A 0.000,B 0.000,C 180.000,E1 0.000} C_DIS
LIN {X 257.744,Y -128.829,Z 420.000,A 0.000,B 0.000,C 180.000,E1 0.000} C_DIS
LIN {X 257.744,Y -128.829,Z 20.000,A 0.000,B 0.000,C 180.000,E1 0.000} C_DIS
LIN {X 257.744,Y -128.829,Z 20.000,A 0.000,B 0.000,C 180.000,E1 0.000} C_DIS
EXTRUDER_STATE=TRUE

;bead-perimeter_outer
$VEL.CP=1
LIN {X 264.034,Y -115.390,Z 20.000,A 0.000,B 0.000,C 180.000,E1 0.000} C_DIS
LIN {X 269.624,Y -101.644,Z 20.000,A 0.000,B 0.000,C 180.000,E1 0.000} C_DIS
LIN {X 274.499,Y -87.629,Z 20.000,A 0.000,B 0.000,C 180.000,E1 0.000} C_DIS
LIN {X 278.646,Y -73.382,Z 20.000,A 0.000,B 0.000,C 180.000,E1 0.000} C_DIS
LIN {X 282.054,Y -58.941,Z 20.000,A 0.000,B 0.000,C 180.000,E1 0.000} C_DIS
LIN {X 284.715,Y -44.343,Z 20.000,A 0.000,B 0.000,C 180.000,E1 0.000} C_DIS
LIN {X 286.619,Y -29.627,Z 20.000,A 0.000,B 0.000,C 180.000,E1 0.000} C_DIS
LIN {X 287.765,Y -14.833,Z 20.000,A 0.000,B 0.000,C 180.000,E1 0.000} C_DIS
LIN {X 288.147,Y 0.000,Z 20.000,A 0.000,B 0.000,C 180.000,E1 0.000} C_DIS
LIN {X 287.765,Y 14.833,Z 20.000,A 0.000,B 0.000,C 180.000,E1 0.000} C_DIS
LIN {X 286.619,Y 29.627,Z 20.000,A 0.000,B 0.000,C 180.000,E1 0.000} C_DIS
LIN {X 284.715,Y 44.343,Z 20.000,A 0.000,B 0.000,C 180.000,E1 0.000} C_DIS
LIN {X 282.054,Y 58.941,Z 20.000,A 0.000,B 0.000,C 180.000,E1 0.000} C_DIS
LIN {X 278.646,Y 73.382,Z 20.000,A 0.000,B 0.000,C 180.000,E1 0.000} C_DIS
LIN {X 274.499,Y 87.629,Z 20.000,A 0.000,B 0.000,C 180.000,E1 0.000} C_DIS
LIN {X 269.624,Y 101.644,Z 20.000,A 0.000,B 0.000,C 180.000,E1 0.000} C_DIS
LIN {X 264.034,Y 115.390,Z 20.000,A 0.000,B 0.000,C 180.000,E1 0.000} C_DIS
LIN {X 257.744,Y 128.829,Z 20.000,A 0.000,B 0.000,C 180.000,E1 0.000} C_DIS
LIN {X 250.770,Y 141.926,Z 20.000,A 0.000,B 0.000,C 180.000,E1 0.000} C_DIS
LIN {X 243.131,Y 154.648,Z 20.000,A 0.000,B 0.000,C 180.000,E1 0.000} C_DIS
LIN {X 234.848,Y 166.958,Z 20.000,A 0.000,B 0.000,C 180.000,E1 0.000} C_DIS
LIN {X 232.107,Y 170.611,Z 20.000,A 0.000,B 0.000,C 180.000,E1 0.000} C_DIS
LIN {X 225.942,Y 178.827,Z 20.000,A 0.000,B 0.000,C 180.000,E1 0.000} C_DIS
LIN {X 216.436,Y 190.221,Z 20.000,A 0.000,B 0.000,C 180.000,E1 0.000} C_DIS
LIN {X 206.357,Y 201.110,Z 20.000,A 0.000,B 0.000,C 180.000,E1 0.000} C_DIS
LIN {X 195.730,Y 211.467,Z 20.000,A 0.000,B 0.000,C 180.000,E1 0.000} C_DIS
LIN {X 184.585,Y 221.262,Z 20.000,A 0.000,B 0.000,C 180.000,E1 0.000} C_DIS
LIN {X 172.949,Y 230.472,Z 20.000,A 0.000,B 0.000,C 180.000,E1 0.000} C_DIS
LIN {X 160.857,Y 239.069,Z 20.000,A 0.000,B 0.000,C 180.000,E1 0.000} C_DIS
LIN {X 148.336,Y 247.033,Z 20.000,A 0.000,B 0.000,C 180.000,E1 0.000} C_DIS
LIN {X 135.422,Y 254.341,Z 20.000,A 0.000,B 0.000,C 180.000,E1 0.000} C_DIS
LIN {X 122.150,Y 260.975,Z 20.000,A 0.000,B 0.000,C 180.000,E1 0.000} C_DIS
LIN {X 108.553,Y 266.916,Z 20.000,A 0.000,B 0.000,C 180.000,E1 0.000} C_DIS
LIN {X 94.668,Y 272.152,Z 20.000,A 0.000,B 0.000,C 180.000,E1 0.000} C_DIS
LIN {X 80.533,Y 276.664,Z 20.000,A 0.000,B 0.000,C 180.000,E1 0.000} C_DIS
LIN {X 66.183,Y 280.443,Z 20.000,A 0.000,B 0.000,C 180.000,E1 0.000} C_DIS
LIN {X 51.659,Y 283.478,Z 20.000,A 0.000,B 0.000,C 180.000,E1 0.000} C_DIS
LIN {X 36.997,Y 285.761,Z 20.000,A 0.000,B 0.000,C 180.000,E1 0.000} C_DIS
LIN {X 22.238,Y 287.287,Z 20.000,A 0.000,B 0.000,C 180.000,E1 0.000} C_DIS
LIN {X 7.419,Y 288.052,Z 20.000,A 0.000,B 0.000,C 180.000,E1 0.000} C_DIS
LIN {X -7.419,Y 288.052,Z 20.000,A 0.000,B 0.000,C 180.000,E1 0.000} C_DIS
LIN {X -22.238,Y 287.287,Z 20.000,A 0.000,B 0.000,C 180.000,E1 0.000} C_DIS
LIN {X -36.997,Y 285.761,Z 20.000,A 0.000,B 0.000,C 180.000,E1 0.000} C_DIS
LIN {X -51.660,Y 283.478,Z 20.000,A 0.000,B 0.000,C 180.000,E1 0.000} C_DIS
LIN {X -66.183,Y 280.443,Z 20.000,A 0.000,B 0.000,C 180.000,E1 0.000} C_DIS
LIN {X -80.533,Y 276.664,Z 20.000,A 0.000,B 0.000,C 180.000,E1 0.000} C_DIS
LIN {X -94.668,Y 272.152,Z 20.000,A 0.000,B 0.000,C 180.000,E1 0.000} C_DIS
LIN {X -108.553,Y 266.916,Z 20.000,A 0.000,B 0.000,C 180.000,E1 0.000} C_DIS
LIN {X -122.150,Y 260.975,Z 20.000,A 0.000,B 0.000,C 180.000,E1 0.000} C_DIS
LIN {X -135.422,Y 254.341,Z 20.000,A 0.000,B 0.000,C 180.000,E1 0.000} C_DIS
LIN {X -148.336,Y 247.033,Z 20.000,A 0.000,B 0.000,C 180.000,E1 0.000} C_DIS
LIN {X -160.857,Y 239.069,Z 20.000,A 0.000,B 0.000,C 180.000,E1 0.000} C_DIS
LIN {X -172.949,Y 230.472,Z 20.000,A 0.000,B 0.000,C 180.000,E1 0.000} C_DIS
LIN {X -184.585,Y 221.262,Z 20.000,A 0.000,B 0.000,C 180.000,E1 0.000} C_DIS
LIN {X -195.730,Y 211.467,Z 20.000,A 0.000,B 0.000,C 180.000,E1 0.000} C_DIS
LIN {X -206.357,Y 201.110,Z 20.000,A 0.000,B 0.000,C 180.000,E1 0.000} C_DIS
LIN {X -216.436,Y 190.221,Z 20.000,A 0.000,B 0.000,C 180.000,E1 0.000} C_DIS
LIN {X -225.942,Y 178.827,Z 20.000,A 0.000,B 0.000,C 180.000,E1 0.000} C_DIS
LIN {X -234.848,Y 166.958,Z 20.000,A 0.000,B 0.000,C 180.000,E1 0.000} C_DIS
LIN {X -243.131,Y 154.648,Z 20.000,A 0.000,B 0.000,C 180.000,E1 0.000} C_DIS
LIN {X -250.770,Y 141.926,Z 20.000,A 0.000,B 0.000,C 180.000,E1 0.000} C_DIS
LIN {X -257.744,Y 128.829,Z 20.000,A 0.000,B 0.000,C 180.000,E1 0.000} C_DIS
LIN {X -264.034,Y 115.390,Z 20.000,A 0.000,B 0.000,C 180.000,E1 0.000} C_DIS
LIN {X -269.624,Y 101.644,Z 20.000,A 0.000,B 0.000,C 180.000,E1 0.000} C_DIS
LIN {X -274.499,Y 87.629,Z 20.000,A 0.000,B 0.000,C 180.000,E1 0.000} C_DIS
LIN {X -278.646,Y 73.382,Z 20.000,A 0.000,B 0.000,C 180.000,E1 0.000} C_DIS
LIN {X -282.054,Y 58.941,Z 20.000,A 0.000,B 0.000,C 180.000,E1 0.000} C_DIS
LIN {X -284.715,Y 44.343,Z 20.000,A 0.000,B 0.000,C 180.000,E1 0.000} C_DIS
LIN {X -286.619,Y 29.627,Z 20.000,A 0.000,B 0.000,C 180.000,E1 0.000} C_DIS
LIN {X -287.765,Y 14.833,Z 20.000,A 0.000,B 0.000,C 180.000,E1 0.000} C_DIS
LIN {X -288.147,Y 0.000,Z 20.000,A 0.000,B 0.000,C 180.000,E1 0.000} C_DIS
LIN {X -287.765,Y -14.833,Z 20.000,A 0.000,B 0.000,C 180.000,E1 0.000} C_DIS
LIN {X -286.619,Y -29.627,Z 20.000,A 0.000,B 0.000,C 180.000,E1 0.000} C_DIS
LIN {X -284.715,Y -44.343,Z 20.000,A 0.000,B 0.000,C 180.000,E1 0.000} C_DIS
LIN {X -282.054,Y -58.941,Z 20.000,A 0.000,B 0.000,C 180.000,E1 0.000} C_DIS
LIN {X -278.646,Y -73.382,Z 20.000,A 0.000,B 0.000,C 180.000,E1 0.000} C_DIS
LIN {X -274.499,Y -87.629,Z 20.000,A 0.000,B 0.000,C 180.000,E1 0.000} C_DIS
LIN {X -269.624,Y -101.644,Z 20.000,A 0.000,B 0.000,C 180.000,E1 0.000} C_DIS
LIN {X -264.034,Y -115.390,Z 20.000,A 0.000,B 0.000,C 180.000,E1 0.000} C_DIS
LIN {X -257.744,Y -128.829,Z 20.000,A 0.000,B 0.000,C 180.000,E1 0.000} C_DIS
LIN {X -250.770,Y -141.926,Z 20.000,A 0.000,B 0.000,C 180.000,E1 0.000} C_DIS
LIN {X -243.131,Y -154.648,Z 20.000,A 0.000,B 0.000,C 180.000,E1 0.000} C_DIS
LIN {X -234.848,Y -166.958,Z 20.000,A 0.000,B 0.000,C 180.000,E1 0.000} C_DIS
LIN {X -225.942,Y -178.827,Z 20.000,A 0.000,B 0.000,C 180.000,E1 0.000} C_DIS
LIN {X -216.436,Y -190.221,Z 20.000,A 0.000,B 0.000,C 180.000,E1 0.000} C_DIS
LIN {X -206.357,Y -201.110,Z 20.000,A 0.000,B 0.000,C 180.000,E1 0.000} C_DIS
LIN {X -195.730,Y -211.467,Z 20.000,A 0.000,B 0.000,C 180.000,E1 0.000} C_DIS
LIN {X -184.585,Y -221.262,Z 20.000,A 0.000,B 0.000,C 180.000,E1 0.000} C_DIS
LIN {X -172.949,Y -230.472,Z 20.000,A 0.000,B 0.000,C 180.000,E1 0.000} C_DIS
LIN {X -160.857,Y -239.069,Z 20.000,A 0.000,B 0.000,C 180.000,E1 0.000} C_DIS
LIN {X -148.336,Y -247.033,Z 20.000,A 0.000,B 0.000,C 180.000,E1 0.000} C_DIS
LIN {X -135.422,Y -254.341,Z 20.000,A 0.000,B 0.000,C 180.000,E1 0.000} C_DIS
LIN {X -122.150,Y -260.975,Z 20.000,A 0.000,B 0.000,C 180.000,E1 0.000} C_DIS
LIN {X -108.553,Y -266.916,Z 20.000,A 0.000,B 0.000,C 180.000,E1 0.000} C_DIS
LIN {X -94.668,Y -272.152,Z 20.000,A 0.000,B 0.000,C 180.000,E1 0.000} C_DIS
LIN {X -80.533,Y -276.664,Z 20.000,A 0.000,B 0.000,C 180.000,E1 0.000} C_DIS
LIN {X -66.183,Y -280.443,Z 20.000,A 0.000,B 0.000,C 180.000,E1 0.000} C_DIS
LIN {X -51.659,Y -283.478,Z 20.000,A 0.000,B 0.000,C 180.000,E1 0.000} C_DIS
LIN {X -36.997,Y -285.761,Z 20.000,A 0.000,B 0.000,C 180.000,E1 0.000} C_DIS
LIN {X -22.238,Y -287.287,Z 20.000,A 0.000,B 0.000,C 180.000,E1 0.000} C_DIS
LIN {X -7.419,Y -288.052,Z 20.000,A 0.000,B 0.000,C 180.000,E1 0.000} C_DIS
LIN {X 7.419,Y -288.052,Z 20.000,A 0.000,B 0.000,C 180.000,E1 0.000} C_DIS
LIN {X 22.238,Y -287.287,Z 20.000,A 0.000,B 0.000,C 180.000,E1 0.000} C_DIS
LIN {X 36.997,Y -285.761,Z 20.000,A 0.000,B 0.000,C 180.000,E1 0.000} C_DIS
LIN {X 51.660,Y -283.478,Z 20.000,A 0.000,B 0.000,C 180.000,E1 0.000} C_DIS
LIN {X 66.183,Y -280.443,Z 20.000,A 0.000,B 0.000,C 180.000,E1 0.000} C_DIS
LIN {X 80.533,Y -276.664,Z 20.000,A 0.000,B 0.000,C 180.000,E1 0.000} C_DIS
LIN {X 94.668,Y -272.152,Z 20.000,A 0.000,B 0.000,C 180.000,E1 0.000} C_DIS
LIN {X 108.553,Y -266.916,Z 20.000,A 0.000,B 0.000,C 180.000,E1 0.000} C_DIS
LIN {X 122.150,Y -260.975,Z 20.000,A 0.000,B 0.000,C 180.000,E1 0.000} C_DIS
LIN {X 135.422,Y -254.341,Z 20.000,A 0.000,B 0.000,C 180.000,E1 0.000} C_DIS
LIN {X 148.336,Y -247.033,Z 20.000,A 0.000,B 0.000,C 180.000,E1 0.000} C_DIS
LIN {X 160.857,Y -239.069,Z 20.000,A 0.000,B 0.000,C 180.000,E1 0.000} C_DIS
LIN {X 172.949,Y -230.472,Z 20.000,A 0.000,B 0.000,C 180.000,E1 0.000} C_DIS
LIN {X 184.585,Y -221.262,Z 20.000,A 0.000,B 0.000,C 180.000,E1 0.000} C_DIS
LIN {X 195.730,Y -211.467,Z 20.000,A 0.000,B 0.000,C 180.000,E1 0.000} C_DIS
LIN {X 206.357,Y -201.110,Z 20.000,A 0.000,B 0.000,C 180.000,E1 0.000} C_DIS
LIN {X 216.436,Y -190.221,Z 20.000,A 0.000,B 0.000,C 180.000,E1 0.000} C_DIS
LIN {X 225.942,Y -178.827,Z 20.000,A 0.000,B 0.000,C 180.000,E1 0.000} C_DIS
LIN {X 234.848,Y -166.958,Z 20.000,A 0.000,B 0.000,C 180.000,E1 0.000} C_DIS
LIN {X 243.131,Y -154.648,Z 20.000,A 0.000,B 0.000,C 180.000,E1 0.000} C_DIS
LIN {X 250.770,Y -141.926,Z 20.000,A 0.000,B 0.000,C 180.000,E1 0.000} C_DIS
LIN {X 257.744,Y -128.829,Z 20.000,A 0.000,B 0.000,C 180.000,E1 0.000} C_DIS
;rapid-leaky
$VEL.CP=0.3
LIN {X 243.839,Y -121.878,Z 20.000,A 0.000,B 0.000,C 180.000,E1 0.000} C_DIS
;bead-perimeter_inner
$VEL.CP=1
LIN {X 249.789,Y -109.164,Z 20.000,A 0.000,B 0.000,C 180.000,E1 0.000} C_DIS
LIN {X 255.078,Y -96.160,Z 20.000,A 0.000,B 0.000,C 180.000,E1 0.000} C_DIS
LIN {X 259.690,Y -82.902,Z 20.000,A 0.000,B 0.000,C 180.000,E1 0.000} C_DIS
LIN {X 263.614,Y -69.424,Z 20.000,A 0.000,B 0.000,C 180.000,E1 0.000} C_DIS
LIN {X 266.838,Y -55.761,Z 20.000,A 0.000,B 0.000,C 180.000,E1 0.000} C_DIS
LIN {X 269.355,Y -41.951,Z 20.000,A 0.000,B 0.000,C 180.000,E1 0.000} C_DIS
LIN {X 271.156,Y -28.029,Z 20.000,A 0.000,B 0.000,C 180.000,E1 0.000} C_DIS
LIN {X 272.241,Y -14.032,Z 20.000,A 0.000,B 0.000,C 180.000,E1 0.000} C_DIS
LIN {X 272.602,Y 0.000,Z 20.000,A 0.000,B 0.000,C 180.000,E1 0.000} C_DIS
LIN {X 272.241,Y 14.032,Z 20.000,A 0.000,B 0.000,C 180.000,E1 0.000} C_DIS
LIN {X 271.156,Y 28.029,Z 20.000,A 0.000,B 0.000,C 180.000,E1 0.000} C_DIS
LIN {X 269.355,Y 41.951,Z 20.000,A 0.000,B 0.000,C 180.000,E1 0.000} C_DIS
LIN {X 266.838,Y 55.761,Z 20.000,A 0.000,B 0.000,C 180.000,E1 0.000} C_DIS
LIN {X 263.614,Y 69.424,Z 20.000,A 0.000,B 0.000,C 180.000,E1 0.000} C_DIS
LIN {X 259.690,Y 82.902,Z 20.000,A 0.000,B 0.000,C 180.000,E1 0.000} C_DIS
LIN {X 255.078,Y 96.160,Z 20.000,A 0.000,B 0.000,C 180.000,E1 0.000} C_DIS
LIN {X 249.789,Y 109.164,Z 20.000,A 0.000,B 0.000,C 180.000,E1 0.000} C_DIS
LIN {X 243.839,Y 121.878,Z 20.000,A 0.000,B 0.000,C 180.000,E1 0.000} C_DIS
LIN {X 237.241,Y 134.269,Z 20.000,A 0.000,B 0.000,C 180.000,E1 0.000} C_DIS
LIN {X 230.014,Y 146.305,Z 20.000,A 0.000,B 0.000,C 180.000,E1 0.000} C_DIS
LIN {X 222.178,Y 157.952,Z 20.000,A 0.000,B 0.000,C 180.000,E1 0.000} C_DIS
LIN {X 219.678,Y 161.284,Z 20.000,A 0.000,B 0.000,C 180.000,E1 0.000} C_DIS
LIN {X 213.753,Y 169.179,Z 20.000,A 0.000,B 0.000,C 180.000,E1 0.000} C_DIS
LIN {X 204.759,Y 179.959,Z 20.000,A 0.000,B 0.000,C 180.000,E1 0.000} C_DIS
LIN {X 195.224,Y 190.261,Z 20.000,A 0.000,B 0.000,C 180.000,E1 0.000} C_DIS
LIN {X 185.170,Y 200.059,Z 20.000,A 0.000,B 0.000,C 180.000,E1 0.000} C_DIS
LIN {X 174.627,Y 209.325,Z 20.000,A 0.000,B 0.000,C 180.000,E1 0.000} C_DIS
LIN {X 163.619,Y 218.038,Z 20.000,A 0.000,B 0.000,C 180.000,E1 0.000} C_DIS
LIN {X 152.179,Y 226.171,Z 20.000,A 0.000,B 0.000,C 180.000,E1 0.000} C_DIS
LIN {X 140.333,Y 233.706,Z 20.000,A 0.000,B 0.000,C 180.000,E1 0.000} C_DIS
LIN {X 128.117,Y 240.620,Z 20.000,A 0.000,B 0.000,C 180.000,E1 0.000} C_DIS
LIN {X 115.561,Y 246.896,Z 20.000,A 0.000,B 0.000,C 180.000,E1 0.000} C_DIS
LIN {X 102.697,Y 252.517,Z 20.000,A 0.000,B 0.000,C 180.000,E1 0.000} C_DIS
LIN {X 89.560,Y 257.470,Z 20.000,A 0.000,B 0.000,C 180.000,E1 0.000} C_DIS
LIN {X 76.188,Y 261.738,Z 20.000,A 0.000,B 0.000,C 180.000,E1 0.000} C_DIS
LIN {X 62.613,Y 265.314,Z 20.000,A 0.000,B 0.000,C 180.000,E1 0.000} C_DIS
LIN {X 48.872,Y 268.185,Z 20.000,A 0.000,B 0.000,C 180.000,E1 0.000} C_DIS
LIN {X 35.002,Y 270.345,Z 20.000,A 0.000,B 0.000,C 180.000,E1 0.000} C_DIS
LIN {X 21.037,Y 271.789,Z 20.000,A 0.000,B 0.000,C 180.000,E1 0.000} C_DIS
LIN {X 7.018,Y 272.512,Z 20.000,A 0.000,B 0.000,C 180.000,E1 0.000} C_DIS
LIN {X -7.018,Y 272.512,Z 20.000,A 0.000,B 0.000,C 180.000,E1 0.000} C_DIS
LIN {X -21.037,Y 271.789,Z 20.000,A 0.000,B 0.000,C 180.000,E1 0.000} C_DIS
LIN {X -35.001,Y 270.345,Z 20.000,A 0.000,B 0.000,C 180.000,E1 0.000} C_DIS
LIN {X -48.873,Y 268.185,Z 20.000,A 0.000,B 0.000,C 180.000,E1 0.000} C_DIS
LIN {X -62.613,Y 265.314,Z 20.000,A 0.000,B 0.000,C 180.000,E1 0.000} C_DIS
LIN {X -76.188,Y 261.738,Z 20.000,A 0.000,B 0.000,C 180.000,E1 0.000} C_DIS
LIN {X -89.560,Y 257.470,Z 20.000,A 0.000,B 0.000,C 180.000,E1 0.000} C_DIS
LIN {X -102.697,Y 252.517,Z 20.000,A 0.000,B 0.000,C 180.000,E1 0.000} C_DIS
LIN {X -115.561,Y 246.896,Z 20.000,A 0.000,B 0.000,C 180.000,E1 0.000} C_DIS
LIN {X -128.117,Y 240.620,Z 20.000,A 0.000,B 0.000,C 180.000,E1 0.000} C_DIS
LIN {X -140.333,Y 233.706,Z 20.000,A 0.000,B 0.000,C 180.000,E1 0.000} C_DIS
LIN {X -152.179,Y 226.171,Z 20.000,A 0.000,B 0.000,C 180.000,E1 0.000} C_DIS
LIN {X -163.619,Y 218.038,Z 20.000,A 0.000,B 0.000,C 180.000,E1 0.000} C_DIS
LIN {X -174.627,Y 209.325,Z 20.000,A 0.000,B 0.000,C 180.000,E1 0.000} C_DIS
LIN {X -185.170,Y 200.059,Z 20.000,A 0.000,B 0.000,C 180.000,E1 0.000} C_DIS
LIN {X -195.225,Y 190.260,Z 20.000,A 0.000,B 0.000,C 180.000,E1 0.000} C_DIS
LIN {X -204.759,Y 179.959,Z 20.000,A 0.000,B 0.000,C 180.000,E1 0.000} C_DIS
LIN {X -213.752,Y 169.179,Z 20.000,A 0.000,B 0.000,C 180.000,E1 0.000} C_DIS
LIN {X -222.178,Y 157.951,Z 20.000,A 0.000,B 0.000,C 180.000,E1 0.000} C_DIS
LIN {X -230.014,Y 146.305,Z 20.000,A 0.000,B 0.000,C 180.000,E1 0.000} C_DIS
LIN {X -237.241,Y 134.269,Z 20.000,A 0.000,B 0.000,C 180.000,E1 0.000} C_DIS
LIN {X -243.839,Y 121.878,Z 20.000,A 0.000,B 0.000,C 180.000,E1 0.000} C_DIS
LIN {X -249.789,Y 109.164,Z 20.000,A 0.000,B 0.000,C 180.000,E1 0.000} C_DIS
LIN {X -255.078,Y 96.160,Z 20.000,A 0.000,B 0.000,C 180.000,E1 0.000} C_DIS
LIN {X -259.690,Y 82.902,Z 20.000,A 0.000,B 0.000,C 180.000,E1 0.000} C_DIS
LIN {X -263.614,Y 69.424,Z 20.000,A 0.000,B 0.000,C 180.000,E1 0.000} C_DIS
LIN {X -266.838,Y 55.761,Z 20.000,A 0.000,B 0.000,C 180.000,E1 0.000} C_DIS
LIN {X -269.355,Y 41.951,Z 20.000,A 0.000,B 0.000,C 180.000,E1 0.000} C_DIS
LIN {X -271.156,Y 28.029,Z 20.000,A 0.000,B 0.000,C 180.000,E1 0.000} C_DIS
LIN {X -272.241,Y 14.032,Z 20.000,A 0.000,B 0.000,C 180.000,E1 0.000} C_DIS
LIN {X -272.602,Y 0.000,Z 20.000,A 0.000,B 0.000,C 180.000,E1 0.000} C_DIS
LIN {X -272.241,Y -14.032,Z 20.000,A 0.000,B 0.000,C 180.000,E1 0.000} C_DIS
LIN {X -271.156,Y -28.029,Z 20.000,A 0.000,B 0.000,C 180.000,E1 0.000} C_DIS
LIN {X -269.355,Y -41.951,Z 20.000,A 0.000,B 0.000,C 180.000,E1 0.000} C_DIS
LIN {X -266.838,Y -55.761,Z 20.000,A 0.000,B 0.000,C 180.000,E1 0.000} C_DIS
LIN {X -263.614,Y -69.424,Z 20.000,A 0.000,B 0.000,C 180.000,E1 0.000} C_DIS
LIN {X -259.690,Y -82.902,Z 20.000,A 0.000,B 0.000,C 180.000,E1 0.000} C_DIS
LIN {X -255.078,Y -96.160,Z 20.000,A 0.000,B 0.000,C 180.000,E1 0.000} C_DIS
LIN {X -249.789,Y -109.164,Z 20.000,A 0.000,B 0.000,C 180.000,E1 0.000} C_DIS
LIN {X -243.839,Y -121.878,Z 20.000,A 0.000,B 0.000,C 180.000,E1 0.000} C_DIS
LIN {X -237.241,Y -134.269,Z 20.000,A 0.000,B 0.000,C 180.000,E1 0.000} C_DIS
LIN {X -230.014,Y -146.305,Z 20.000,A 0.000,B 0.000,C 180.000,E1 0.000} C_DIS
LIN {X -222.178,Y -157.952,Z 20.000,A 0.000,B 0.000,C 180.000,E1 0.000} C_DIS
LIN {X -213.753,Y -169.179,Z 20.000,A 0.000,B 0.000,C 180.000,E1 0.000} C_DIS
LIN {X -204.759,Y -179.959,Z 20.000,A 0.000,B 0.000,C 180.000,E1 0.000} C_DIS
LIN {X -195.224,Y -190.261,Z 20.000,A 0.000,B 0.000,C 180.000,E1 0.000} C_DIS
LIN {X -185.170,Y -200.059,Z 20.000,A 0.000,B 0.000,C 180.000,E1 0.000} C_DIS
LIN {X -174.627,Y -209.325,Z 20.000,A 0.000,B 0.000,C 180.000,E1 0.000} C_DIS
LIN {X -163.619,Y -218.038,Z 20.000,A 0.000,B 0.000,C 180.000,E1 0.000} C_DIS
LIN {X -152.179,Y -226.171,Z 20.000,A 0.000,B 0.000,C 180.000,E1 0.000} C_DIS
LIN {X -140.333,Y -233.706,Z 20.000,A 0.000,B 0.000,C 180.000,E1 0.000} C_DIS
LIN {X -128.117,Y -240.620,Z 20.000,A 0.000,B 0.000,C 180.000,E1 0.000} C_DIS
LIN {X -115.561,Y -246.896,Z 20.000,A 0.000,B 0.000,C 180.000,E1 0.000} C_DIS
LIN {X -102.697,Y -252.517,Z 20.000,A 0.000,B 0.000,C 180.000,E1 0.000} C_DIS
LIN {X -89.560,Y -257.470,Z 20.000,A 0.000,B 0.000,C 180.000,E1 0.000} C_DIS
LIN {X -76.188,Y -261.738,Z 20.000,A 0.000,B 0.000,C 180.000,E1 0.000} C_DIS
LIN {X -62.613,Y -265.314,Z 20.000,A 0.000,B 0.000,C 180.000,E1 0.000} C_DIS
LIN {X -48.872,Y -268.185,Z 20.000,A 0.000,B 0.000,C 180.000,E1 0.000} C_DIS
LIN {X -35.002,Y -270.345,Z 20.000,A 0.000,B 0.000,C 180.000,E1 0.000} C_DIS
LIN {X -21.037,Y -271.789,Z 20.000,A 0.000,B 0.000,C 180.000,E1 0.000} C_DIS
LIN {X -7.018,Y -272.512,Z 20.000,A 0.000,B 0.000,C 180.000,E1 0.000} C_DIS
LIN {X 7.018,Y -272.512,Z 20.000,A 0.000,B 0.000,C 180.000,E1 0.000} C_DIS
LIN {X 21.037,Y -271.789,Z 20.000,A 0.000,B 0.000,C 180.000,E1 0.000} C_DIS
LIN {X 35.001,Y -270.345,Z 20.000,A 0.000,B 0.000,C 180.000,E1 0.000} C_DIS
LIN {X 48.873,Y -268.185,Z 20.000,A 0.000,B 0.000,C 180.000,E1 0.000} C_DIS
LIN {X 62.613,Y -265.314,Z 20.000,A 0.000,B 0.000,C 180.000,E1 0.000} C_DIS
LIN {X 76.188,Y -261.738,Z 20.000,A 0.000,B 0.000,C 180.000,E1 0.000} C_DIS
LIN {X 89.560,Y -257.470,Z 20.000,A 0.000,B 0.000,C 180.000,E1 0.000} C_DIS
LIN {X 102.697,Y -252.517,Z 20.000,A 0.000,B 0.000,C 180.000,E1 0.000} C_DIS
LIN {X 115.561,Y -246.896,Z 20.000,A 0.000,B 0.000,C 180.000,E1 0.000} C_DIS
LIN {X 128.117,Y -240.620,Z 20.000,A 0.000,B 0.000,C 180.000,E1 0.000} C_DIS
LIN {X 140.333,Y -233.706,Z 20.000,A 0.000,B 0.000,C 180.000,E1 0.000} C_DIS
LIN {X 152.179,Y -226.171,Z 20.000,A 0.000,B 0.000,C 180.000,E1 0.000} C_DIS
LIN {X 163.619,Y -218.038,Z 20.000,A 0.000,B 0.000,C 180.000,E1 0.000} C_DIS
LIN {X 174.627,Y -209.325,Z 20.000,A 0.000,B 0.000,C 180.000,E1 0.000} C_DIS
LIN {X 185.170,Y -200.059,Z 20.000,A 0.000,B 0.000,C 180.000,E1 0.000} C_DIS
LIN {X 195.225,Y -190.260,Z 20.000,A 0.000,B 0.000,C 180.000,E1 0.000} C_DIS
LIN {X 204.759,Y -179.959,Z 20.000,A 0.000,B 0.000,C 180.000,E1 0.000} C_DIS
LIN {X 213.752,Y -169.179,Z 20.000,A 0.000,B 0.000,C 180.000,E1 0.000} C_DIS
LIN {X 222.178,Y -157.951,Z 20.000,A 0.000,B 0.000,C 180.000,E1 0.000} C_DIS
LIN {X 230.014,Y -146.305,Z 20.000,A 0.000,B 0.000,C 180.000,E1 0.000} C_DIS
LIN {X 237.241,Y -134.269,Z 20.000,A 0.000,B 0.000,C 180.000,E1 0.000} C_DIS
LIN {X 243.839,Y -121.878,Z 20.000,A 0.000,B 0.000,C 180.000,E1 0.000} C_DIS
;rapid-leaky
$VEL.CP=0.3
LIN {X 224.032,Y -121.288,Z 20.000,A 0.000,B 0.000,C 180.000,E1 0.000} C_DIS
;bead-solid_infill
$VEL.CP=1
LIN {X 121.185,Y -224.136,Z 20.000,A 0.000,B 0.000,C 180.000,E1 0.000} C_DIS
LIN {X 119.767,Y -224.938,Z 20.000,A 0.000,B 0.000,C 180.000,E1 0.000} C_DIS
LIN {X 108.030,Y -230.805,Z 20.000,A 0.000,B 0.000,C 180.000,E1 0.000} C_DIS
LIN {X 99.254,Y -234.640,Z 20.000,A 0.000,B 0.000,C 180.000,E1 0.000} C_DIS
LIN {X 96.004,Y -236.059,Z 20.000,A 0.000,B 0.000,C 180.000,E1 0.000} C_DIS
LIN {X 83.723,Y -240.690,Z 20.000,A 0.000,B 0.000,C 180.000,E1 0.000} C_DIS
LIN {X 71.223,Y -244.680,Z 20.000,A 0.000,B 0.000,C 180.000,E1 0.000} C_DIS
LIN {X 68.538,Y -245.387,Z 20.000,A 0.000,B 0.000,C 180.000,E1 0.000} C_DIS
LIN {X 245.369,Y -68.556,Z 20.000,A 0.000,B 0.000,C 180.000,E1 0.000} C_DIS
LIN {X 246.434,Y -64.899,Z 20.000,A 0.000,B 0.000,C 180.000,E1 0.000} C_DIS
LIN {X 249.447,Y -52.127,Z 20.000,A 0.000,B 0.000,C 180.000,E1 0.000} C_DIS
LIN {X 251.800,Y -39.218,Z 20.000,A 0.000,B 0.000,C 180.000,E1 0.000} C_DIS
LIN {X 253.062,Y -29.467,Z 20.000,A 0.000,B 0.000,C 180.000,E1 0.000} C_DIS
LIN {X 29.467,Y -253.062,Z 20.000,A 0.000,B 0.000,C 180.000,E1 0.000} C_DIS
LIN {X 19.665,Y -254.076,Z 20.000,A 0.000,B 0.000,C 180.000,E1 0.000} C_DIS
LIN {X 6.560,Y -254.752,Z 20.000,A 0.000,B 0.000,C 180.000,E1 0.000} C_DIS
LIN {X -3.618,Y -254.752,Z 20.000,A 0.000,B 0.000,C 180.000,E1 0.000} C_DIS
LIN {X 254.743,Y 3.609,Z 20.000,A 0.000,B 0.000,C 180.000,E1 0.000} C_DIS
LIN {X 254.498,Y 13.117,Z 20.000,A 0.000,B 0.000,C 180.000,E1 0.000} C_DIS
LIN {X 253.485,Y 26.202,Z 20.000,A 0.000,B 0.000,C 180.000,E1 0.000} C_DIS
LIN {X 252.620,Y 32.882,Z 20.000,A 0.000,B 0.000,C 180.000,E1 0.000} C_DIS
LIN {X -32.951,Y -252.690,Z 20.000,A 0.000,B 0.000,C 180.000,E1 0.000} C_DIS
LIN {X -45.688,Y -250.707,Z 20.000,A 0.000,B 0.000,C 180.000,E1 0.000} C_DIS
LIN {X -58.532,Y -248.023,Z 20.000,A 0.000,B 0.000,C 180.000,E1 0.000} C_DIS
LIN {X -59.440,Y -247.784,Z 20.000,A 0.000,B 0.000,C 180.000,E1 0.000} C_DIS
LIN {X 247.733,Y 59.391,Z 20.000,A 0.000,B 0.000,C 180.000,E1 0.000} C_DIS
LIN {X 246.434,Y 64.899,Z 20.000,A 0.000,B 0.000,C 180.000,E1 0.000} C_DIS
LIN {X 242.766,Y 77.499,Z 20.000,A 0.000,B 0.000,C 180.000,E1 0.000} C_DIS
LIN {X 240.619,Y 83.672,Z 20.000,A 0.000,B 0.000,C 180.000,E1 0.000} C_DIS
LIN {X -83.737,Y -240.685,Z 20.000,A 0.000,B 0.000,C 180.000,E1 0.000} C_DIS
LIN {X -96.004,Y -236.059,Z 20.000,A 0.000,B 0.000,C 180.000,E1 0.000} C_DIS
LIN {X -106.097,Y -231.649,Z 20.000,A 0.000,B 0.000,C 180.000,E1 0.000} C_DIS
LIN {X 231.626,Y 106.075,Z 20.000,A 0.000,B 0.000,C 180.000,E1 0.000} C_DIS
LIN {X 227.948,Y 113.935,Z 20.000,A 0.000,B 0.000,C 180.000,E1 0.000} C_DIS
LIN {X 225.073,Y 119.334,Z 20.000,A 0.000,B 0.000,C 180.000,E1 0.000} C_DIS
LIN {X 221.780,Y 125.518,Z 20.000,A 0.000,B 0.000,C 180.000,E1 0.000} C_DIS
LIN {X 220.990,Y 126.834,Z 20.000,A 0.000,B 0.000,C 180.000,E1 0.000} C_DIS
LIN {X -126.801,Y -220.957,Z 20.000,A 0.000,B 0.000,C 180.000,E1 0.000} C_DIS
LIN {X -131.187,Y -218.475,Z 20.000,A 0.000,B 0.000,C 180.000,E1 0.000} C_DIS
LIN {X -142.261,Y -211.431,Z 20.000,A 0.000,B 0.000,C 180.000,E1 0.000} C_DIS
LIN {X -146.007,Y -208.768,Z 20.000,A 0.000,B 0.000,C 180.000,E1 0.000} C_DIS
LIN {X 208.792,Y 146.032,Z 20.000,A 0.000,B 0.000,C 180.000,E1 0.000} C_DIS
LIN {X 207.698,Y 147.658,Z 20.000,A 0.000,B 0.000,C 180.000,E1 0.000} C_DIS
LIN {X 205.473,Y 150.624,Z 20.000,A 0.000,B 0.000,C 180.000,E1 0.000} C_DIS
LIN {X 199.822,Y 158.153,Z 20.000,A 0.000,B 0.000,C 180.000,E1 0.000} C_DIS
LIN {X 195.136,Y 163.771,Z 20.000,A 0.000,B 0.000,C 180.000,E1 0.000} C_DIS
LIN {X -163.816,Y -195.182,Z 20.000,A 0.000,B 0.000,C 180.000,E1 0.000} C_DIS
LIN {X -173.103,Y -187.020,Z 20.000,A 0.000,B 0.000,C 180.000,E1 0.000} C_DIS
LIN {X -180.166,Y -180.136,Z 20.000,A 0.000,B 0.000,C 180.000,E1 0.000} C_DIS
LIN {X 180.136,Y 180.166,Z 20.000,A 0.000,B 0.000,C 180.000,E1 0.000} C_DIS
LIN {X 173.103,Y 187.020,Z 20.000,A 0.000,B 0.000,C 180.000,E1 0.000} C_DIS
LIN {X 163.784,Y 195.210,Z 20.000,A 0.000,B 0.000,C 180.000,E1 0.000} C_DIS
LIN {X -195.163,Y -163.737,Z 20.000,A 0.000,B 0.000,C 180.000,E1 0.000} C_DIS
LIN {X -199.821,Y -158.154,Z 20.000,A 0.000,B 0.000,C 180.000,E1 0.000} C_DIS
LIN {X -207.699,Y -147.658,Z 20.000,A 0.000,B 0.000,C 180.000,E1 0.000} C_DIS
LIN {X -208.817,Y -145.996,Z 20.000,A 0.000,B 0.000,C 180.000,E1 0.000} C_DIS
LIN {X 145.972,Y 208.793,Z 20.000,A 0.000,B 0.000,C 180.000,E1 0.000} C_DIS
LIN {X 142.261,Y 211.431,Z 20.000,A 0.000,B 0.000,C 180.000,E1 0.000} C_DIS
LIN {X 131.187,Y 218.475,Z 20.000,A 0.000,B 0.000,C 180.000,E1 0.000} C_DIS
LIN {X 126.762,Y 220.979,Z 20.000,A 0.000,B 0.000,C 180.000,E1 0.000} C_DIS
LIN {X -221.013,Y -126.796,Z 20.000,A 0.000,B 0.000,C 180.000,E1 0.000} C_DIS
LIN {X -221.780,Y -125.518,Z 20.000,A 0.000,B 0.000,C 180.000,E1 0.000} C_DIS
LIN {X -224.675,Y -120.082,Z 20.000,A 0.000,B 0.000,C 180.000,E1 0.000} C_DIS
LIN {X -227.948,Y -113.935,Z 20.000,A 0.000,B 0.000,C 180.000,E1 0.000} C_DIS
LIN {X -231.646,Y -106.033,Z 20.000,A 0.000,B 0.000,C 180.000,E1 0.000} C_DIS
LIN {X 106.055,Y 231.668,Z 20.000,A 0.000,B 0.000,C 180.000,E1 0.000} C_DIS
LIN {X 96.004,Y 236.059,Z 20.000,A 0.000,B 0.000,C 180.000,E1 0.000} C_DIS
LIN {X 83.723,Y 240.690,Z 20.000,A 0.000,B 0.000,C 180.000,E1 0.000} C_DIS
LIN {X 83.692,Y 240.700,Z 20.000,A 0.000,B 0.000,C 180.000,E1 0.000} C_DIS
LIN {X -240.634,Y -83.627,Z 20.000,A 0.000,B 0.000,C 180.000,E1 0.000} C_DIS
LIN {X -242.766,Y -77.499,Z 20.000,A 0.000,B 0.000,C 180.000,E1 0.000} C_DIS
LIN {X -246.434,Y -64.899,Z 20.000,A 0.000,B 0.000,C 180.000,E1 0.000} C_DIS
LIN {X -247.745,Y -59.342,Z 20.000,A 0.000,B 0.000,C 180.000,E1 0.000} C_DIS
LIN {X 59.392,Y 247.796,Z 20.000,A 0.000,B 0.000,C 180.000,E1 0.000} C_DIS
LIN {X 58.532,Y 248.023,Z 20.000,A 0.000,B 0.000,C 180.000,E1 0.000} C_DIS
LIN {X 45.688,Y 250.707,Z 20.000,A 0.000,B 0.000,C 180.000,E1 0.000} C_DIS
LIN {X 32.899,Y 252.698,Z 20.000,A 0.000,B 0.000,C 180.000,E1 0.000} C_DIS
LIN {X -252.627,Y -32.828,Z 20.000,A 0.000,B 0.000,C 180.000,E1 0.000} C_DIS
LIN {X -253.485,Y -26.202,Z 20.000,A 0.000,B 0.000,C 180.000,E1 0.000} C_DIS
LIN {X -254.498,Y -13.117,Z 20.000,A 0.000,B 0.000,C 180.000,E1 0.000} C_DIS
LIN {X -254.745,Y -3.550,Z 20.000,A 0.000,B 0.000,C 180.000,E1 0.000} C_DIS
LIN {X 3.557,Y 254.752,Z 20.000,A 0.000,B 0.000,C 180.000,E1 0.000} C_DIS
LIN {X -6.560,Y 254.752,Z 20.000,A 0.000,B 0.000,C 180.000,E1 0.000} C_DIS
LIN {X -19.665,Y 254.076,Z 20.000,A 0.000,B 0.000,C 180.000,E1 0.000} C_DIS
LIN {X -29.535,Y 253.055,Z 20.000,A 0.000,B 0.000,C 180.000,E1 0.000} C_DIS
LIN {X -253.053,Y 29.537,Z 20.000,A 0.000,B 0.000,C 180.000,E1 0.000} C_DIS
LIN {X -251.800,Y 39.218,Z 20.000,A 0.000,B 0.000,C 180.000,E1 0.000} C_DIS
LIN {X -249.447,Y 52.127,Z 20.000,A 0.000,B 0.000,C 180.000,E1 0.000} C_DIS
LIN {X -247.338,Y 61.068,Z 20.000,A 0.000,B 0.000,C 180.000,E1 0.000} C_DIS
LIN {X -246.434,Y 64.899,Z 20.000,A 0.000,B 0.000,C 180.000,E1 0.000} C_DIS
LIN {X -245.344,Y 68.641,Z 20.000,A 0.000,B 0.000,C 180.000,E1 0.000} C_DIS
LIN {X -68.620,Y 245.366,Z 20.000,A 0.000,B 0.000,C 180.000,E1 0.000} C_DIS
LIN {X -71.223,Y 244.680,Z 20.000,A 0.000,B 0.000,C 180.000,E1 0.000} C_DIS
LIN {X -83.723,Y 240.690,Z 20.000,A 0.000,B 0.000,C 180.000,E1 0.000} C_DIS
LIN {X -96.004,Y 236.059,Z 20.000,A 0.000,B 0.000,C 180.000,E1 0.000} C_DIS
LIN {X -99.253,Y 234.640,Z 20.000,A 0.000,B 0.000,C 180.000,E1 0.000} C_DIS
LIN {X -108.030,Y 230.805,Z 20.000,A 0.000,B 0.000,C 180.000,E1 0.000} C_DIS
LIN {X -119.767,Y 224.938,Z 20.000,A 0.000,B 0.000,C 180.000,E1 0.000} C_DIS
LIN {X -121.325,Y 224.056,Z 20.000,A 0.000,B 0.000,C 180.000,E1 0.000} C_DIS
LIN {X -223.963,Y 121.418,Z 20.000,A 0.000,B 0.000,C 180.000,E1 0.000} C_DIS
$VEL.CP=0.3
LIN {X -223.963,Y 121.418,Z 20.000,A 0.000,B 0.000,C 180.000,E1 0.000} C_DIS
EXTRUDER_STATE=FALSE

LIN {X 44.590,Y -175.026,Z 430.000,A 0.000,B 0.000,C 180.000,E1 0.000} C_DIS
LIN {X 121.828,Y -260.287,Z 430.000,A 0.000,B 0.000,C 180.000,E1 0.000} C_DIS
LIN {X 121.828,Y -260.287,Z 30.000,A 0.000,B 0.000,C 180.000,E1 0.000} C_DIS
LIN {X 121.828,Y -260.287,Z 30.000,A 0.000,B 0.000,C 180.000,E1 0.000} C_DIS
EXTRUDER_STATE=TRUE
;bead-perimeter_outer
$VEL.CP=1
LIN {X 135.066,Y -253.671,Z 30.000,A 0.000,B 0.000,C 180.000,E1 0.000} C_DIS
LIN {X 147.945,Y -246.382,Z 30.000,A 0.000,B 0.000,C 180.000,E1 0.000} C_DIS
LIN {X 160.432,Y -238.439,Z 30.000,A 0.000,B 0.000,C 180.000,E1 0.000} C_DIS
LIN {X 172.493,Y -229.864,Z 30.000,A 0.000,B 0.000,C 180.000,E1 0.000} C_DIS
LIN {X 184.098,Y -220.679,Z 30.000,A 0.000,B 0.000,C 180.000,E1 0.000} C_DIS
LIN {X 195.215,Y -210.909,Z 30.000,A 0.000,B 0.000,C 180.000,E1 0.000} C_DIS
LIN {X 205.813,Y -200.580,Z 30.000,A 0.000,B 0.000,C 180.000,E1 0.000} C_DIS
LIN {X 215.866,Y -189.720,Z 30.000,A 0.000,B 0.000,C 180.000,E1 0.000} C_DIS
LIN {X 225.346,Y -178.356,Z 30.000,A 0.000,B 0.000,C 180.000,E1 0.000} C_DIS
LIN {X 234.229,Y -166.518,Z 30.000,A 0.000,B 0.000,C 180.000,E1 0.000} C_DIS
LIN {X 242.491,Y -154.240,Z 30.000,A 0.000,B 0.000,C 180.000,E1 0.000} C_DIS
LIN {X 250.109,Y -141.552,Z 30.000,A 0.000,B 0.000,C 180.000,E1 0.000} C_DIS
LIN {X 257.064,Y -128.489,Z 30.000,A 0.000,B 0.000,C 180.000,E1 0.000} C_DIS
LIN {X 263.339,Y -115.085,Z 30.000,A 0.000,B 0.000,C 180.000,E1 0.000} C_DIS
LIN {X 268.913,Y -101.377,Z 30.000,A 0.000,B 0.000,C 180.000,E1 0.000} C_DIS
LIN {X 273.773,Y -87.405,Z 30.000,A 0.000,B 0.000,C 180.000,E1 0.000} C_DIS
LIN {X 277.911,Y -73.189,Z 30.000,A 0.000,B 0.000,C 180.000,E1 0.000} C_DIS
LIN {X 281.311,Y -58.786,Z 30.000,A 0.000,B 0.000,C 180.000,E1 0.000} C_DIS
LIN {X 283.964,Y -44.226,Z 30.000,A 0.000,B 0.000,C 180.000,E1 0.000} C_DIS
LIN {X 285.864,Y -29.549,Z 30.000,A 0.000,B 0.000,C 180.000,E1 0.000} C_DIS
LIN {X 287.006,Y -14.794,Z 30.000,A 0.000,B 0.000,C 180.000,E1 0.000} C_DIS
LIN {X 287.387,Y 0.000,Z 30.000,A 0.000,B 0.000,C 180.000,E1 0.000} C_DIS
LIN {X 287.006,Y 14.794,Z 30.000,A 0.000,B 0.000,C 180.000,E1 0.000} C_DIS
LIN {X 285.864,Y 29.549,Z 30.000,A 0.000,B 0.000,C 180.000,E1 0.000} C_DIS
LIN {X 283.964,Y 44.226,Z 30.000,A 0.000,B 0.000,C 180.000,E1 0.000} C_DIS
LIN {X 281.311,Y 58.786,Z 30.000,A 0.000,B 0.000,C 180.000,E1 0.000} C_DIS
LIN {X 277.942,Y 73.063,Z 30.000,A 0.000,B 0.000,C 180.000,E1 0.000} C_DIS
LIN {X 273.775,Y 87.398,Z 30.000,A 0.000,B 0.000,C 180.000,E1 0.000} C_DIS
LIN {X 268.913,Y 101.377,Z 30.000,A 0.000,B 0.000,C 180.000,E1 0.000} C_DIS
LIN {X 263.339,Y 115.085,Z 30.000,A 0.000,B 0.000,C 180.000,E1 0.000} C_DIS
LIN {X 257.064,Y 128.489,Z 30.000,A 0.000,B 0.000,C 180.000,E1 0.000} C_DIS
LIN {X 250.109,Y 141.552,Z 30.000,A 0.000,B 0.000,C 180.000,E1 0.000} C_DIS
LIN {X 242.491,Y 154.240,Z 30.000,A 0.000,B 0.000,C 180.000,E1 0.000} C_DIS
LIN {X 234.229,Y 166.518,Z 30.000,A 0.000,B 0.000,C 180.000,E1 0.000} C_DIS
LIN {X 225.346,Y 178.356,Z 30.000,A 0.000,B 0.000,C 180.000,E1 0.000} C_DIS
LIN {X 215.866,Y 189.720,Z 30.000,A 0.000,B 0.000,C 180.000,E1 0.000} C_DIS
LIN {X 205.813,Y 200.580,Z 30.000,A 0.000,B 0.000,C 180.000,E1 0.000} C_DIS
LIN {X 195.215,Y 210.909,Z 30.000,A 0.000,B 0.000,C 180.000,E1 0.000} C_DIS
LIN {X 184.098,Y 220.679,Z 30.000,A 0.000,B 0.000,C 180.000,E1 0.000} C_DIS
LIN {X 172.493,Y 229.864,Z 30.000,A 0.000,B 0.000,C 180.000,E1 0.000} C_DIS
LIN {X 160.432,Y 238.439,Z 30.000,A 0.000,B 0.000,C 180.000,E1 0.000} C_DIS
LIN {X 147.945,Y 246.382,Z 30.000,A 0.000,B 0.000,C 180.000,E1 0.000} C_DIS
LIN {X 135.066,Y 253.671,Z 30.000,A 0.000,B 0.000,C 180.000,E1 0.000} C_DIS
LIN {X 121.828,Y 260.287,Z 30.000,A 0.000,B 0.000,C 180.000,E1 0.000} C_DIS
LIN {X 108.266,Y 266.213,Z 30.000,A 0.000,B 0.000,C 180.000,E1 0.000} C_DIS
LIN {X 94.419,Y 271.435,Z 30.000,A 0.000,B 0.000,C 180.000,E1 0.000} C_DIS
LIN {X 80.321,Y 275.935,Z 30.000,A 0.000,B 0.000,C 180.000,E1 0.000} C_DIS
LIN {X 66.010,Y 279.704,Z 30.000,A 0.000,B 0.000,C 180.000,E1 0.000} C_DIS
LIN {X 51.523,Y 282.731,Z 30.000,A 0.000,B 0.000,C 180.000,E1 0.000} C_DIS
LIN {X 36.900,Y 285.008,Z 30.000,A 0.000,B 0.000,C 180.000,E1 0.000} C_DIS
LIN {X 22.179,Y 286.530,Z 30.000,A 0.000,B 0.000,C 180.000,E1 0.000} C_DIS
LIN {X 7.400,Y 287.292,Z 30.000,A 0.000,B 0.000,C 180.000,E1 0.000} C_DIS
LIN {X -7.400,Y 287.292,Z 30.000,A 0.000,B 0.000,C 180.000,E1 0.000} C_DIS
LIN {X -22.177,Y 286.531,Z 30.000,A 0.000,B 0.000,C 180.000,E1 0.000} C_DIS
LIN {X -36.900,Y 285.008,Z 30.000,A 0.000,B 0.000,C 180.000,E1 0.000} C_DIS
LIN {X -51.523,Y 282.731,Z 30.000,A 0.000,B 0.000,C 180.000,E1 0.000} C_DIS
LIN {X -66.010,Y 279.704,Z 30.000,A 0.000,B 0.000,C 180.000,E1 0.000} C_DIS
LIN {X -80.321,Y 275.935,Z 30.000,A 0.000,B 0.000,C 180.000,E1 0.000} C_DIS
LIN {X -94.419,Y 271.435,Z 30.000,A 0.000,B 0.000,C 180.000,E1 0.000} C_DIS
LIN {X -108.266,Y 266.213,Z 30.000,A 0.000,B 0.000,C 180.000,E1 0.000} C_DIS
LIN {X -121.828,Y 260.287,Z 30.000,A 0.000,B 0.000,C 180.000,E1 0.000} C_DIS
LIN {X -135.066,Y 253.671,Z 30.000,A 0.000,B 0.000,C 180.000,E1 0.000} C_DIS
LIN {X -147.945,Y 246.382,Z 30.000,A 0.000,B 0.000,C 180.000,E1 0.000} C_DIS
LIN {X -160.432,Y 238.439,Z 30.000,A 0.000,B 0.000,C 180.000,E1 0.000} C_DIS
LIN {X -172.493,Y 229.864,Z 30.000,A 0.000,B 0.000,C 180.000,E1 0.000} C_DIS
LIN {X -184.098,Y 220.679,Z 30.000,A 0.000,B 0.000,C 180.000,E1 0.000} C_DIS
LIN {X -195.215,Y 210.909,Z 30.000,A 0.000,B 0.000,C 180.000,E1 0.000} C_DIS
LIN {X -205.813,Y 200.580,Z 30.000,A 0.000,B 0.000,C 180.000,E1 0.000} C_DIS
LIN {X -215.866,Y 189.720,Z 30.000,A 0.000,B 0.000,C 180.000,E1 0.000} C_DIS
LIN {X -225.346,Y 178.356,Z 30.000,A 0.000,B 0.000,C 180.000,E1 0.000} C_DIS
LIN {X -234.229,Y 166.518,Z 30.000,A 0.000,B 0.000,C 180.000,E1 0.000} C_DIS
LIN {X -242.491,Y 154.240,Z 30.000,A 0.000,B 0.000,C 180.000,E1 0.000} C_DIS
LIN {X -250.109,Y 141.552,Z 30.000,A 0.000,B 0.000,C 180.000,E1 0.000} C_DIS
LIN {X -257.064,Y 128.489,Z 30.000,A 0.000,B 0.000,C 180.000,E1 0.000} C_DIS
LIN {X -263.339,Y 115.085,Z 30.000,A 0.000,B 0.000,C 180.000,E1 0.000} C_DIS
LIN {X -268.913,Y 101.377,Z 30.000,A 0.000,B 0.000,C 180.000,E1 0.000} C_DIS
LIN {X -273.773,Y 87.405,Z 30.000,A 0.000,B 0.000,C 180.000,E1 0.000} C_DIS
LIN {X -277.911,Y 73.189,Z 30.000,A 0.000,B 0.000,C 180.000,E1 0.000} C_DIS
LIN {X -281.311,Y 58.786,Z 30.000,A 0.000,B 0.000,C 180.000,E1 0.000} C_DIS
LIN {X -283.964,Y 44.226,Z 30.000,A 0.000,B 0.000,C 180.000,E1 0.000} C_DIS
LIN {X -285.864,Y 29.549,Z 30.000,A 0.000,B 0.000,C 180.000,E1 0.000} C_DIS
LIN {X -287.006,Y 14.794,Z 30.000,A 0.000,B 0.000,C 180.000,E1 0.000} C_DIS
LIN {X -287.387,Y 0.000,Z 30.000,A 0.000,B 0.000,C 180.000,E1 0.000} C_DIS
LIN {X -287.006,Y -14.794,Z 30.000,A 0.000,B 0.000,C 180.000,E1 0.000} C_DIS
LIN {X -285.864,Y -29.549,Z 30.000,A 0.000,B 0.000,C 180.000,E1 0.000} C_DIS
LIN {X -283.964,Y -44.226,Z 30.000,A 0.000,B 0.000,C 180.000,E1 0.000} C_DIS
LIN {X -281.311,Y -58.786,Z 30.000,A 0.000,B 0.000,C 180.000,E1 0.000} C_DIS
LIN {X -277.914,Y -73.179,Z 30.000,A 0.000,B 0.000,C 180.000,E1 0.000} C_DIS
LIN {X -273.775,Y -87.398,Z 30.000,A 0.000,B 0.000,C 180.000,E1 0.000} C_DIS
LIN {X -268.913,Y -101.377,Z 30.000,A 0.000,B 0.000,C 180.000,E1 0.000} C_DIS
LIN {X -263.339,Y -115.085,Z 30.000,A 0.000,B 0.000,C 180.000,E1 0.000} C_DIS
LIN {X -257.064,Y -128.489,Z 30.000,A 0.000,B 0.000,C 180.000,E1 0.000} C_DIS
LIN {X -250.109,Y -141.552,Z 30.000,A 0.000,B 0.000,C 180.000,E1 0.000} C_DIS
LIN {X -242.491,Y -154.240,Z 30.000,A 0.000,B 0.000,C 180.000,E1 0.000} C_DIS
LIN {X -234.229,Y -166.518,Z 30.000,A 0.000,B 0.000,C 180.000,E1 0.000} C_DIS
LIN {X -225.346,Y -178.356,Z 30.000,A 0.000,B 0.000,C 180.000,E1 0.000} C_DIS
LIN {X -215.866,Y -189.720,Z 30.000,A 0.000,B 0.000,C 180.000,E1 0.000} C_DIS
LIN {X -205.813,Y -200.580,Z 30.000,A 0.000,B 0.000,C 180.000,E1 0.000} C_DIS
LIN {X -195.215,Y -210.909,Z 30.000,A 0.000,B 0.000,C 180.000,E1 0.000} C_DIS
LIN {X -184.098,Y -220.679,Z 30.000,A 0.000,B 0.000,C 180.000,E1 0.000} C_DIS
LIN {X -172.493,Y -229.864,Z 30.000,A 0.000,B 0.000,C 180.000,E1 0.000} C_DIS
LIN {X -160.432,Y -238.439,Z 30.000,A 0.000,B 0.000,C 180.000,E1 0.000} C_DIS
LIN {X -147.945,Y -246.382,Z 30.000,A 0.000,B 0.000,C 180.000,E1 0.000} C_DIS
LIN {X -135.066,Y -253.671,Z 30.000,A 0.000,B 0.000,C 180.000,E1 0.000} C_DIS
LIN {X -121.828,Y -260.287,Z 30.000,A 0.000,B 0.000,C 180.000,E1 0.000} C_DIS
LIN {X -108.266,Y -266.213,Z 30.000,A 0.000,B 0.000,C 180.000,E1 0.000} C_DIS
LIN {X -94.419,Y -271.435,Z 30.000,A 0.000,B 0.000,C 180.000,E1 0.000} C_DIS
LIN {X -80.321,Y -275.935,Z 30.000,A 0.000,B 0.000,C 180.000,E1 0.000} C_DIS
LIN {X -66.010,Y -279.704,Z 30.000,A 0.000,B 0.000,C 180.000,E1 0.000} C_DIS
LIN {X -51.523,Y -282.731,Z 30.000,A 0.000,B 0.000,C 180.000,E1 0.000} C_DIS
LIN {X -36.900,Y -285.008,Z 30.000,A 0.000,B 0.000,C 180.000,E1 0.000} C_DIS
LIN {X -22.179,Y -286.530,Z 30.000,A 0.000,B 0.000,C 180.000,E1 0.000} C_DIS
LIN {X -7.400,Y -287.292,Z 30.000,A 0.000,B 0.000,C 180.000,E1 0.000} C_DIS
LIN {X 7.400,Y -287.292,Z 30.000,A 0.000,B 0.000,C 180.000,E1 0.000} C_DIS
LIN {X 22.177,Y -286.531,Z 30.000,A 0.000,B 0.000,C 180.000,E1 0.000} C_DIS
LIN {X 36.900,Y -285.008,Z 30.000,A 0.000,B 0.000,C 180.000,E1 0.000} C_DIS
LIN {X 51.523,Y -282.731,Z 30.000,A 0.000,B 0.000,C 180.000,E1 0.000} C_DIS
LIN {X 66.010,Y -279.704,Z 30.000,A 0.000,B 0.000,C 180.000,E1 0.000} C_DIS
LIN {X 80.321,Y -275.935,Z 30.000,A 0.000,B 0.000,C 180.000,E1 0.000} C_DIS
LIN {X 94.419,Y -271.435,Z 30.000,A 0.000,B 0.000,C 180.000,E1 0.000} C_DIS
LIN {X 108.266,Y -266.213,Z 30.000,A 0.000,B 0.000,C 180.000,E1 0.000} C_DIS
LIN {X 121.828,Y -260.287,Z 30.000,A 0.000,B 0.000,C 180.000,E1 0.000} C_DIS
;rapid-leaky
$VEL.CP=0.3
LIN {X 115.239,Y -246.208,Z 30.000,A 0.000,B 0.000,C 180.000,E1 0.000} C_DIS
;bead-perimeter_inner
$VEL.CP=1
LIN {X 127.760,Y -239.950,Z 30.000,A 0.000,B 0.000,C 180.000,E1 0.000} C_DIS
LIN {X 139.942,Y -233.055,Z 30.000,A 0.000,B 0.000,C 180.000,E1 0.000} C_DIS
LIN {X 151.754,Y -225.541,Z 30.000,A 0.000,B 0.000,C 180.000,E1 0.000} C_DIS
LIN {X 163.163,Y -217.430,Z 30.000,A 0.000,B 0.000,C 180.000,E1 0.000} C_DIS
LIN {X 174.140,Y -208.742,Z 30.000,A 0.000,B 0.000,C 180.000,E1 0.000} C_DIS
LIN {X 184.655,Y -199.501,Z 30.000,A 0.000,B 0.000,C 180.000,E1 0.000} C_DIS
LIN {X 194.681,Y -189.730,Z 30.000,A 0.000,B 0.000,C 180.000,E1 0.000} C_DIS
LIN {X 204.190,Y -179.457,Z 30.000,A 0.000,B 0.000,C 180.000,E1 0.000} C_DIS
LIN {X 213.157,Y -168.708,Z 30.000,A 0.000,B 0.000,C 180.000,E1 0.000} C_DIS
LIN {X 221.559,Y -157.511,Z 30.000,A 0.000,B 0.000,C 180.000,E1 0.000} C_DIS
LIN {X 229.374,Y -145.897,Z 30.000,A 0.000,B 0.000,C 180.000,E1 0.000} C_DIS
LIN {X 236.580,Y -133.896,Z 30.000,A 0.000,B 0.000,C 180.000,E1 0.000} C_DIS
LIN {X 243.159,Y -121.539,Z 30.000,A 0.000,B 0.000,C 180.000,E1 0.000} C_DIS
LIN {X 249.094,Y -108.860,Z 30.000,A 0.000,B 0.000,C 180.000,E1 0.000} C_DIS
LIN {X 254.367,Y -95.894,Z 30.000,A 0.000,B 0.000,C 180.000,E1 0.000} C_DIS
LIN {X 258.964,Y -82.680,Z 30.000,A 0.000,B 0.000,C 180.000,E1 0.000} C_DIS
LIN {X 262.879,Y -69.230,Z 30.000,A 0.000,B 0.000,C 180.000,E1 0.000} C_DIS
LIN {X 266.095,Y -55.606,Z 30.000,A 0.000,B 0.000,C 180.000,E1 0.000} C_DIS
LIN {X 268.604,Y -41.834,Z 30.000,A 0.000,B 0.000,C 180.000,E1 0.000} C_DIS
LIN {X 270.401,Y -27.951,Z 30.000,A 0.000,B 0.000,C 180.000,E1 0.000} C_DIS
LIN {X 271.482,Y -13.994,Z 30.000,A 0.000,B 0.000,C 180.000,E1 0.000} C_DIS
LIN {X 271.842,Y 0.000,Z 30.000,A 0.000,B 0.000,C 180.000,E1 0.000} C_DIS
LIN {X 271.482,Y 13.994,Z 30.000,A 0.000,B 0.000,C 180.000,E1 0.000} C_DIS
LIN {X 270.401,Y 27.951,Z 30.000,A 0.000,B 0.000,C 180.000,E1 0.000} C_DIS
LIN {X 268.604,Y 41.834,Z 30.000,A 0.000,B 0.000,C 180.000,E1 0.000} C_DIS
LIN {X 266.094,Y 55.607,Z 30.000,A 0.000,B 0.000,C 180.000,E1 0.000} C_DIS
LIN {X 262.883,Y 69.217,Z 30.000,A 0.000,B 0.000,C 180.000,E1 0.000} C_DIS
LIN {X 258.966,Y 82.671,Z 30.000,A 0.000,B 0.000,C 180.000,E1 0.000} C_DIS
LIN {X 254.367,Y 95.894,Z 30.000,A 0.000,B 0.000,C 180.000,E1 0.000} C_DIS
LIN {X 249.094,Y 108.860,Z 30.000,A 0.000,B 0.000,C 180.000,E1 0.000} C_DIS
LIN {X 243.159,Y 121.539,Z 30.000,A 0.000,B 0.000,C 180.000,E1 0.000} C_DIS
LIN {X 236.580,Y 133.896,Z 30.000,A 0.000,B 0.000,C 180.000,E1 0.000} C_DIS
LIN {X 229.374,Y 145.897,Z 30.000,A 0.000,B 0.000,C 180.000,E1 0.000} C_DIS
LIN {X 221.559,Y 157.511,Z 30.000,A 0.000,B 0.000,C 180.000,E1 0.000} C_DIS
LIN {X 213.157,Y 168.708,Z 30.000,A 0.000,B 0.000,C 180.000,E1 0.000} C_DIS
LIN {X 204.190,Y 179.457,Z 30.000,A 0.000,B 0.000,C 180.000,E1 0.000} C_DIS
LIN {X 194.681,Y 189.730,Z 30.000,A 0.000,B 0.000,C 180.000,E1 0.000} C_DIS
LIN {X 184.655,Y 199.501,Z 30.000,A 0.000,B 0.000,C 180.000,E1 0.000} C_DIS
LIN {X 174.140,Y 208.742,Z 30.000,A 0.000,B 0.000,C 180.000,E1 0.000} C_DIS
LIN {X 163.163,Y 217.430,Z 30.000,A 0.000,B 0.000,C 180.000,E1 0.000} C_DIS
LIN {X 151.754,Y 225.541,Z 30.000,A 0.000,B 0.000,C 180.000,E1 0.000} C_DIS
LIN {X 139.942,Y 233.055,Z 30.000,A 0.000,B 0.000,C 180.000,E1 0.000} C_DIS
LIN {X 127.760,Y 239.950,Z 30.000,A 0.000,B 0.000,C 180.000,E1 0.000} C_DIS
LIN {X 115.239,Y 246.208,Z 30.000,A 0.000,B 0.000,C 180.000,E1 0.000} C_DIS
LIN {X 102.409,Y 251.814,Z 30.000,A 0.000,B 0.000,C 180.000,E1 0.000} C_DIS
LIN {X 89.311,Y 256.753,Z 30.000,A 0.000,B 0.000,C 180.000,E1 0.000} C_DIS
LIN {X 75.976,Y 261.009,Z 30.000,A 0.000,B 0.000,C 180.000,E1 0.000} C_DIS
LIN {X 62.439,Y 264.575,Z 30.000,A 0.000,B 0.000,C 180.000,E1 0.000} C_DIS
LIN {X 48.736,Y 267.438,Z 30.000,A 0.000,B 0.000,C 180.000,E1 0.000} C_DIS
LIN {X 34.904,Y 269.592,Z 30.000,A 0.000,B 0.000,C 180.000,E1 0.000} C_DIS
LIN {X 20.979,Y 271.032,Z 30.000,A 0.000,B 0.000,C 180.000,E1 0.000} C_DIS
LIN {X 7.000,Y 271.752,Z 30.000,A 0.000,B 0.000,C 180.000,E1 0.000} C_DIS
LIN {X -7.000,Y 271.752,Z 30.000,A 0.000,B 0.000,C 180.000,E1 0.000} C_DIS
LIN {X -20.977,Y 271.032,Z 30.000,A 0.000,B 0.000,C 180.000,E1 0.000} C_DIS
LIN {X -34.904,Y 269.592,Z 30.000,A 0.000,B 0.000,C 180.000,E1 0.000} C_DIS
LIN {X -48.736,Y 267.438,Z 30.000,A 0.000,B 0.000,C 180.000,E1 0.000} C_DIS
LIN {X -62.439,Y 264.575,Z 30.000,A 0.000,B 0.000,C 180.000,E1 0.000} C_DIS
LIN {X -75.976,Y 261.009,Z 30.000,A 0.000,B 0.000,C 180.000,E1 0.000} C_DIS
LIN {X -89.311,Y 256.753,Z 30.000,A 0.000,B 0.000,C 180.000,E1 0.000} C_DIS
LIN {X -102.409,Y 251.814,Z 30.000,A 0.000,B 0.000,C 180.000,E1 0.000} C_DIS
LIN {X -115.239,Y 246.208,Z 30.000,A 0.000,B 0.000,C 180.000,E1 0.000} C_DIS
LIN {X -127.760,Y 239.950,Z 30.000,A 0.000,B 0.000,C 180.000,E1 0.000} C_DIS
LIN {X -139.942,Y 233.055,Z 30.000,A 0.000,B 0.000,C 180.000,E1 0.000} C_DIS
LIN {X -151.754,Y 225.541,Z 30.000,A 0.000,B 0.000,C 180.000,E1 0.000} C_DIS
LIN {X -163.163,Y 217.430,Z 30.000,A 0.000,B 0.000,C 180.000,E1 0.000} C_DIS
LIN {X -174.140,Y 208.742,Z 30.000,A 0.000,B 0.000,C 180.000,E1 0.000} C_DIS
LIN {X -184.655,Y 199.501,Z 30.000,A 0.000,B 0.000,C 180.000,E1 0.000} C_DIS
LIN {X -194.681,Y 189.730,Z 30.000,A 0.000,B 0.000,C 180.000,E1 0.000} C_DIS
LIN {X -204.190,Y 179.457,Z 30.000,A 0.000,B 0.000,C 180.000,E1 0.000} C_DIS
LIN {X -213.157,Y 168.708,Z 30.000,A 0.000,B 0.000,C 180.000,E1 0.000} C_DIS
LIN {X -221.559,Y 157.511,Z 30.000,A 0.000,B 0.000,C 180.000,E1 0.000} C_DIS
LIN {X -229.374,Y 145.897,Z 30.000,A 0.000,B 0.000,C 180.000,E1 0.000} C_DIS
LIN {X -236.580,Y 133.896,Z 30.000,A 0.000,B 0.000,C 180.000,E1 0.000} C_DIS
LIN {X -243.159,Y 121.539,Z 30.000,A 0.000,B 0.000,C 180.000,E1 0.000} C_DIS
LIN {X -249.094,Y 108.860,Z 30.000,A 0.000,B 0.000,C 180.000,E1 0.000} C_DIS
LIN {X -254.367,Y 95.894,Z 30.000,A 0.000,B 0.000,C 180.000,E1 0.000} C_DIS
LIN {X -258.964,Y 82.680,Z 30.000,A 0.000,B 0.000,C 180.000,E1 0.000} C_DIS
LIN {X -262.879,Y 69.230,Z 30.000,A 0.000,B 0.000,C 180.000,E1 0.000} C_DIS
LIN {X -266.095,Y 55.606,Z 30.000,A 0.000,B 0.000,C 180.000,E1 0.000} C_DIS
LIN {X -268.604,Y 41.834,Z 30.000,A 0.000,B 0.000,C 180.000,E1 0.000} C_DIS
LIN {X -270.401,Y 27.951,Z 30.000,A 0.000,B 0.000,C 180.000,E1 0.000} C_DIS
LIN {X -271.482,Y 13.994,Z 30.000,A 0.000,B 0.000,C 180.000,E1 0.000} C_DIS
LIN {X -271.842,Y 0.000,Z 30.000,A 0.000,B 0.000,C 180.000,E1 0.000} C_DIS
LIN {X -271.482,Y -13.994,Z 30.000,A 0.000,B 0.000,C 180.000,E1 0.000} C_DIS
LIN {X -270.401,Y -27.951,Z 30.000,A 0.000,B 0.000,C 180.000,E1 0.000} C_DIS
LIN {X -268.604,Y -41.834,Z 30.000,A 0.000,B 0.000,C 180.000,E1 0.000} C_DIS
LIN {X -266.094,Y -55.607,Z 30.000,A 0.000,B 0.000,C 180.000,E1 0.000} C_DIS
LIN {X -262.883,Y -69.217,Z 30.000,A 0.000,B 0.000,C 180.000,E1 0.000} C_DIS
LIN {X -258.966,Y -82.671,Z 30.000,A 0.000,B 0.000,C 180.000,E1 0.000} C_DIS
LIN {X -254.367,Y -95.894,Z 30.000,A 0.000,B 0.000,C 180.000,E1 0.000} C_DIS
LIN {X -249.094,Y -108.860,Z 30.000,A 0.000,B 0.000,C 180.000,E1 0.000} C_DIS
LIN {X -243.159,Y -121.539,Z 30.000,A 0.000,B 0.000,C 180.000,E1 0.000} C_DIS
LIN {X -236.580,Y -133.896,Z 30.000,A 0.000,B 0.000,C 180.000,E1 0.000} C_DIS
LIN {X -229.374,Y -145.897,Z 30.000,A 0.000,B 0.000,C 180.000,E1 0.000} C_DIS
LIN {X -221.559,Y -157.511,Z 30.000,A 0.000,B 0.000,C 180.000,E1 0.000} C_DIS
LIN {X -213.157,Y -168.708,Z 30.000,A 0.000,B 0.000,C 180.000,E1 0.000} C_DIS
LIN {X -204.190,Y -179.457,Z 30.000,A 0.000,B 0.000,C 180.000,E1 0.000} C_DIS
LIN {X -194.681,Y -189.730,Z 30.000,A 0.000,B 0.000,C 180.000,E1 0.000} C_DIS
LIN {X -184.655,Y -199.501,Z 30.000,A 0.000,B 0.000,C 180.000,E1 0.000} C_DIS
LIN {X -174.140,Y -208.742,Z 30.000,A 0.000,B 0.000,C 180.000,E1 0.000} C_DIS
LIN {X -163.163,Y -217.430,Z 30.000,A 0.000,B 0.000,C 180.000,E1 0.000} C_DIS
LIN {X -151.754,Y -225.541,Z 30.000,A 0.000,B 0.000,C 180.000,E1 0.000} C_DIS
LIN {X -139.942,Y -233.055,Z 30.000,A 0.000,B 0.000,C 180.000,E1 0.000} C_DIS
LIN {X -127.760,Y -239.950,Z 30.000,A 0.000,B 0.000,C 180.000,E1 0.000} C_DIS
LIN {X -115.239,Y -246.208,Z 30.000,A 0.000,B 0.000,C 180.000,E1 0.000} C_DIS
LIN {X -102.409,Y -251.814,Z 30.000,A 0.000,B 0.000,C 180.000,E1 0.000} C_DIS
LIN {X -89.311,Y -256.753,Z 30.000,A 0.000,B 0.000,C 180.000,E1 0.000} C_DIS
LIN {X -75.976,Y -261.009,Z 30.000,A 0.000,B 0.000,C 180.000,E1 0.000} C_DIS
LIN {X -62.439,Y -264.575,Z 30.000,A 0.000,B 0.000,C 180.000,E1 0.000} C_DIS
LIN {X -48.736,Y -267.438,Z 30.000,A 0.000,B 0.000,C 180.000,E1 0.000} C_DIS
LIN {X -34.904,Y -269.592,Z 30.000,A 0.000,B 0.000,C 180.000,E1 0.000} C_DIS
LIN {X -20.979,Y -271.032,Z 30.000,A 0.000,B 0.000,C 180.000,E1 0.000} C_DIS
LIN {X -7.000,Y -271.752,Z 30.000,A 0.000,B 0.000,C 180.000,E1 0.000} C_DIS
LIN {X 7.000,Y -271.752,Z 30.000,A 0.000,B 0.000,C 180.000,E1 0.000} C_DIS
LIN {X 20.977,Y -271.032,Z 30.000,A 0.000,B 0.000,C 180.000,E1 0.000} C_DIS
LIN {X 34.904,Y -269.592,Z 30.000,A 0.000,B 0.000,C 180.000,E1 0.000} C_DIS
LIN {X 48.736,Y -267.438,Z 30.000,A 0.000,B 0.000,C 180.000,E1 0.000} C_DIS
LIN {X 62.439,Y -264.575,Z 30.000,A 0.000,B 0.000,C 180.000,E1 0.000} C_DIS
LIN {X 75.976,Y -261.009,Z 30.000,A 0.000,B 0.000,C 180.000,E1 0.000} C_DIS
LIN {X 89.311,Y -256.753,Z 30.000,A 0.000,B 0.000,C 180.000,E1 0.000} C_DIS
LIN {X 102.409,Y -251.814,Z 30.000,A 0.000,B 0.000,C 180.000,E1 0.000} C_DIS
LIN {X 115.239,Y -246.208,Z 30.000,A 0.000,B 0.000,C 180.000,E1 0.000} C_DIS
$VEL.CP=0.3
LIN {X 115.239,Y -246.208,Z 30.000,A 0.000,B 0.000,C 180.000,E1 0.000} C_DIS
EXTRUDER_STATE=FALSE

LIN {X -282.725,Y -205.906,Z 430.000,A 0.000,B 0.000,C 180.000,E1 0.000} C_DIS
LIN {X -123.334,Y -222.047,Z 430.000,A 0.000,B 0.000,C 180.000,E1 0.000} C_DIS
LIN {X -123.334,Y -222.047,Z 30.000,A 0.000,B 0.000,C 180.000,E1 0.000} C_DIS
LIN {X -123.334,Y -222.047,Z 30.000,A 0.000,B 0.000,C 180.000,E1 0.000} C_DIS
EXTRUDER_STATE=TRUE

;bead-solid_infill
$VEL.CP=1
LIN {X -222.123,Y -123.259,Z 30.000,A 0.000,B 0.000,C 180.000,E1 0.000} C_DIS
LIN {X -227.268,Y -113.595,Z 30.000,A 0.000,B 0.000,C 180.000,E1 0.000} C_DIS
LIN {X -232.815,Y -101.746,Z 30.000,A 0.000,B 0.000,C 180.000,E1 0.000} C_DIS
LIN {X -237.743,Y -89.628,Z 30.000,A 0.000,B 0.000,C 180.000,E1 0.000} C_DIS
LIN {X -242.042,Y -77.268,Z 30.000,A 0.000,B 0.000,C 180.000,E1 0.000} C_DIS
LIN {X -244.228,Y -69.758,Z 30.000,A 0.000,B 0.000,C 180.000,E1 0.000} C_DIS
LIN {X -69.685,Y -244.300,Z 30.000,A 0.000,B 0.000,C 180.000,E1 0.000} C_DIS
LIN {X -58.359,Y -247.284,Z 30.000,A 0.000,B 0.000,C 180.000,E1 0.000} C_DIS
LIN {X -45.551,Y -249.960,Z 30.000,A 0.000,B 0.000,C 180.000,E1 0.000} C_DIS
LIN {X -32.623,Y -251.973,Z 30.000,A 0.000,B 0.000,C 180.000,E1 0.000} C_DIS
LIN {X -30.386,Y -252.204,Z 30.000,A 0.000,B 0.000,C 180.000,E1 0.000} C_DIS
LIN {X -252.174,Y -30.417,Z 30.000,A 0.000,B 0.000,C 180.000,E1 0.000} C_DIS
LIN {X -252.730,Y -26.124,Z 30.000,A 0.000,B 0.000,C 180.000,E1 0.000} C_DIS
LIN {X -253.739,Y -13.080,Z 30.000,A 0.000,B 0.000,C 180.000,E1 0.000} C_DIS
LIN {X -254.076,Y 0.000,Z 30.000,A 0.000,B 0.000,C 180.000,E1 0.000} C_DIS
LIN {X -254.004,Y 2.809,Z 30.000,A 0.000,B 0.000,C 180.000,E1 0.000} C_DIS
LIN {X 2.797,Y -253.992,Z 30.000,A 0.000,B 0.000,C 180.000,E1 0.000} C_DIS
LIN {X 6.543,Y -253.992,Z 30.000,A 0.000,B 0.000,C 180.000,E1 0.000} C_DIS
LIN {X 19.606,Y -253.319,Z 30.000,A 0.000,B 0.000,C 180.000,E1 0.000} C_DIS
LIN {X 32.216,Y -252.015,Z 30.000,A 0.000,B 0.000,C 180.000,E1 0.000} C_DIS
LIN {X -251.949,Y 32.150,Z 30.000,A 0.000,B 0.000,C 180.000,E1 0.000} C_DIS
LIN {X -251.049,Y 39.100,Z 30.000,A 0.000,B 0.000,C 180.000,E1 0.000} C_DIS
LIN {X -248.704,Y 51.972,Z 30.000,A 0.000,B 0.000,C 180.000,E1 0.000} C_DIS
LIN {X -247.114,Y 58.710,Z 30.000,A 0.000,B 0.000,C 180.000,E1 0.000} C_DIS
LIN {X 58.772,Y -247.175,Z 30.000,A 0.000,B 0.000,C 180.000,E1 0.000} C_DIS
LIN {X 71.011,Y -243.951,Z 30.000,A 0.000,B 0.000,C 180.000,E1 0.000} C_DIS
LIN {X 83.088,Y -240.096,Z 30.000,A 0.000,B 0.000,C 180.000,E1 0.000} C_DIS
LIN {X -240.038,Y 83.030,Z 30.000,A 0.000,B 0.000,C 180.000,E1 0.000} C_DIS
LIN {X -237.743,Y 89.627,Z 30.000,A 0.000,B 0.000,C 180.000,E1 0.000} C_DIS
LIN {X -232.815,Y 101.746,Z 30.000,A 0.000,B 0.000,C 180.000,E1 0.000} C_DIS
LIN {X -231.075,Y 105.462,Z 30.000,A 0.000,B 0.000,C 180.000,E1 0.000} C_DIS
LIN {X 105.479,Y -231.091,Z 30.000,A 0.000,B 0.000,C 180.000,E1 0.000} C_DIS
LIN {X 107.708,Y -230.117,Z 30.000,A 0.000,B 0.000,C 180.000,E1 0.000} C_DIS
LIN {X 119.410,Y -224.268,Z 30.000,A 0.000,B 0.000,C 180.000,E1 0.000} C_DIS
LIN {X 126.205,Y -220.422,Z 30.000,A 0.000,B 0.000,C 180.000,E1 0.000} C_DIS
LIN {X -220.460,Y 126.242,Z 30.000,A 0.000,B 0.000,C 180.000,E1 0.000} C_DIS
LIN {X -214.383,Y 136.363,Z 30.000,A 0.000,B 0.000,C 180.000,E1 0.000} C_DIS
LIN {X -208.270,Y 145.448,Z 30.000,A 0.000,B 0.000,C 180.000,E1 0.000} C_DIS
LIN {X 145.427,Y -208.248,Z 30.000,A 0.000,B 0.000,C 180.000,E1 0.000} C_DIS
LIN {X 152.499,Y -203.221,Z 30.000,A 0.000,B 0.000,C 180.000,E1 0.000} C_DIS
LIN {X 157.944,Y -198.911,Z 30.000,A 0.000,B 0.000,C 180.000,E1 0.000} C_DIS
LIN {X 162.759,Y -195.100,Z 30.000,A 0.000,B 0.000,C 180.000,E1 0.000} C_DIS
LIN {X 163.246,Y -194.672,Z 30.000,A 0.000,B 0.000,C 180.000,E1 0.000} C_DIS
LIN {X -194.625,Y 163.199,Z 30.000,A 0.000,B 0.000,C 180.000,E1 0.000} C_DIS
LIN {X -190.845,Y 167.729,Z 30.000,A 0.000,B 0.000,C 180.000,E1 0.000} C_DIS
LIN {X -181.958,Y 177.331,Z 30.000,A 0.000,B 0.000,C 180.000,E1 0.000} C_DIS
LIN {X -179.630,Y 179.599,Z 30.000,A 0.000,B 0.000,C 180.000,E1 0.000} C_DIS
LIN {X 179.599,Y -179.629,Z 30.000,A 0.000,B 0.000,C 180.000,E1 0.000} C_DIS
LIN {X 181.958,Y -177.331,Z 30.000,A 0.000,B 0.000,C 180.000,E1 0.000} C_DIS
LIN {X 190.845,Y -167.729,Z 30.000,A 0.000,B 0.000,C 180.000,E1 0.000} C_DIS
LIN {X 194.597,Y -163.232,Z 30.000,A 0.000,B 0.000,C 180.000,E1 0.000} C_DIS
LIN {X -163.279,Y 194.643,Z 30.000,A 0.000,B 0.000,C 180.000,E1 0.000} C_DIS
LIN {X -162.759,Y 195.100,Z 30.000,A 0.000,B 0.000,C 180.000,E1 0.000} C_DIS
LIN {X -152.499,Y 203.221,Z 30.000,A 0.000,B 0.000,C 180.000,E1 0.000} C_DIS
LIN {X -145.463,Y 208.223,Z 30.000,A 0.000,B 0.000,C 180.000,E1 0.000} C_DIS
LIN {X 208.246,Y -145.485,Z 30.000,A 0.000,B 0.000,C 180.000,E1 0.000} C_DIS
LIN {X 214.383,Y -136.363,Z 30.000,A 0.000,B 0.000,C 180.000,E1 0.000} C_DIS
LIN {X 220.437,Y -126.280,Z 30.000,A 0.000,B 0.000,C 180.000,E1 0.000} C_DIS
LIN {X -126.244,Y 220.400,Z 30.000,A 0.000,B 0.000,C 180.000,E1 0.000} C_DIS
LIN {X -119.410,Y 224.268,Z 30.000,A 0.000,B 0.000,C 180.000,E1 0.000} C_DIS
LIN {X -107.708,Y 230.117,Z 30.000,A 0.000,B 0.000,C 180.000,E1 0.000} C_DIS
LIN {X -105.521,Y 231.073,Z 30.000,A 0.000,B 0.000,C 180.000,E1 0.000} C_DIS
LIN {X 231.056,Y -105.504,Z 30.000,A 0.000,B 0.000,C 180.000,E1 0.000} C_DIS
LIN {X 232.815,Y -101.746,Z 30.000,A 0.000,B 0.000,C 180.000,E1 0.000} C_DIS
LIN {X 237.743,Y -89.627,Z 30.000,A 0.000,B 0.000,C 180.000,E1 0.000} C_DIS
LIN {X 240.022,Y -83.075,Z 30.000,A 0.000,B 0.000,C 180.000,E1 0.000} C_DIS
LIN {X -83.134,Y 240.081,Z 30.000,A 0.000,B 0.000,C 180.000,E1 0.000} C_DIS
LIN {X -71.011,Y 243.951,Z 30.000,A 0.000,B 0.000,C 180.000,E1 0.000} C_DIS
LIN {X -58.820,Y 247.162,Z 30.000,A 0.000,B 0.000,C 180.000,E1 0.000} C_DIS
LIN {X 247.102,Y -58.759,Z 30.000,A 0.000,B 0.000,C 180.000,E1 0.000} C_DIS
LIN {X 248.704,Y -51.972,Z 30.000,A 0.000,B 0.000,C 180.000,E1 0.000} C_DIS
LIN {X 251.049,Y -39.100,Z 30.000,A 0.000,B 0.000,C 180.000,E1 0.000} C_DIS
LIN {X 251.942,Y -32.204,Z 30.000,A 0.000,B 0.000,C 180.000,E1 0.000} C_DIS
LIN {X -32.271,Y 252.009,Z 30.000,A 0.000,B 0.000,C 180.000,E1 0.000} C_DIS
LIN {X -19.606,Y 253.319,Z 30.000,A 0.000,B 0.000,C 180.000,E1 0.000} C_DIS
LIN {X -6.543,Y 253.992,Z 30.000,A 0.000,B 0.000,C 180.000,E1 0.000} C_DIS
LIN {X -2.858,Y 253.992,Z 30.000,A 0.000,B 0.000,C 180.000,E1 0.000} C_DIS
LIN {X 254.002,Y -2.868,Z 30.000,A 0.000,B 0.000,C 180.000,E1 0.000} C_DIS
LIN {X 254.076,Y 0.000,Z 30.000,A 0.000,B 0.000,C 180.000,E1 0.000} C_DIS
LIN {X 253.739,Y 13.080,Z 30.000,A 0.000,B 0.000,C 180.000,E1 0.000} C_DIS
LIN {X 252.730,Y 26.124,Z 30.000,A 0.000,B 0.000,C 180.000,E1 0.000} C_DIS
LIN {X 252.183,Y 30.347,Z 30.000,A 0.000,B 0.000,C 180.000,E1 0.000} C_DIS
LIN {X 30.318,Y 252.211,Z 30.000,A 0.000,B 0.000,C 180.000,E1 0.000} C_DIS
LIN {X 32.623,Y 251.973,Z 30.000,A 0.000,B 0.000,C 180.000,E1 0.000} C_DIS
LIN {X 45.551,Y 249.960,Z 30.000,A 0.000,B 0.000,C 180.000,E1 0.000} C_DIS
LIN {X 58.359,Y 247.284,Z 30.000,A 0.000,B 0.000,C 180.000,E1 0.000} C_DIS
LIN {X 69.603,Y 244.322,Z 30.000,A 0.000,B 0.000,C 180.000,E1 0.000} C_DIS
LIN {X 244.253,Y 69.672,Z 30.000,A 0.000,B 0.000,C 180.000,E1 0.000} C_DIS
LIN {X 242.042,Y 77.268,Z 30.000,A 0.000,B 0.000,C 180.000,E1 0.000} C_DIS
LIN {X 237.743,Y 89.628,Z 30.000,A 0.000,B 0.000,C 180.000,E1 0.000} C_DIS
LIN {X 232.815,Y 101.746,Z 30.000,A 0.000,B 0.000,C 180.000,E1 0.000} C_DIS
LIN {X 227.268,Y 113.595,Z 30.000,A 0.000,B 0.000,C 180.000,E1 0.000} C_DIS
LIN {X 222.192,Y 123.129,Z 30.000,A 0.000,B 0.000,C 180.000,E1 0.000} C_DIS
LIN {X 123.194,Y 222.126,Z 30.000,A 0.000,B 0.000,C 180.000,E1 0.000} C_DIS
$VEL.CP=0.3
LIN {X 123.194,Y 222.126,Z 30.000,A 0.000,B 0.000,C 180.000,E1 0.000} C_DIS
EXTRUDER_STATE=FALSE

LIN {X -28.198,Y -148.117,Z 440.000,A 0.000,B 0.000,C 180.000,E1 0.000} C_DIS
LIN {X -79.969,Y -274.726,Z 440.000,A 0.000,B 0.000,C 180.000,E1 0.000} C_DIS
LIN {X -79.969,Y -274.726,Z 40.000,A 0.000,B 0.000,C 180.000,E1 0.000} C_DIS
LIN {X -79.969,Y -274.726,Z 40.000,A 0.000,B 0.000,C 180.000,E1 0.000} C_DIS
EXTRUDER_STATE=TRUE

